// ---- DUTs/IO/PDOs/InfoData_6F19DB2B.TcDUT
{attribute 'GeneratedUsingTerminal: EK1100-0000-0018'}
{attribute addProperty BoxType "EK1100-0000-0018"}
{attribute addProperty Id "StateAT %I*UINT2"}
{attribute addProperty CRC "1863965483"}
{attribute addProperty Size "2"}
TYPE InfoData_6F19DB2B :
STRUCT
	{attribute addProperty Name "State"}
	State AT %I* : UINT;
END_STRUCT
END_TYPE

// ---- DUTs/IO/PDOs/YVR_Inputs_4719D0DB.TcDUT
{attribute 'GeneratedUsingTerminal: APS1003-7000-0016'}
{attribute addProperty BoxType "APS1003-7000-0016"}
{attribute addProperty Id "StatusWordAT %I*UINT2Current_D_0X0AT %I*INT2Current_D_0X1AT %I*INT2Current_D_0X2AT %I*INT2Current_D_0Y0AT %I*INT2Current_D_0Y1AT %I*INT2Current_D_0Y2AT %I*INT2Current_D_1X0AT %I*INT2Current_D_1X1AT %I*INT2Current_D_1X2AT %I*INT2Current_D_1Y0AT %I*INT2Current_D_1Y1AT %I*INT2Current_D_1Y2AT %I*INT2Current_D_2X0AT %I*INT2Current_D_2X1AT %I*INT2Current_D_2X2AT %I*INT2Current_D_2Y0AT %I*INT2Current_D_2Y1AT %I*INT2Current_D_2Y2AT %I*INT2Current_D_3X0AT %I*INT2Current_D_3X1AT %I*INT2Current_D_3X2AT %I*INT2Current_D_3Y0AT %I*INT2Current_D_3Y1AT %I*INT2Current_D_3Y2AT %I*INT2Current_Q_0X0AT %I*INT2Current_Q_0X1AT %I*INT2Current_Q_0X2AT %I*INT2Current_Q_0Y0AT %I*INT2Current_Q_0Y1AT %I*INT2Current_Q_0Y2AT %I*INT2Current_Q_1X0AT %I*INT2Current_Q_1X1AT %I*INT2Current_Q_1X2AT %I*INT2Current_Q_1Y0AT %I*INT2Current_Q_1Y1AT %I*INT2Current_Q_1Y2AT %I*INT2Current_Q_2X0AT %I*INT2Current_Q_2X1AT %I*INT2Current_Q_2X2AT %I*INT2Current_Q_2Y0AT %I*INT2Current_Q_2Y1AT %I*INT2Current_Q_2Y2AT %I*INT2Current_Q_3X0AT %I*INT2Current_Q_3X1AT %I*INT2Current_Q_3X2AT %I*INT2Current_Q_3Y0AT %I*INT2Current_Q_3Y1AT %I*INT2Current_Q_3Y2AT %I*INT2"}
{attribute addProperty CRC "1192874203"}
{attribute addProperty Size "98"}
TYPE YVR_Inputs_4719D0DB EXTENDS InputBase_8311D824 :
STRUCT
	{attribute addProperty Name "StatusWord"}
	StatusWord AT %I* : UINT;
	{attribute addProperty Name "Current_D_0X0"}
	Current_D_0X0 AT %I* : INT;
	{attribute addProperty Name "Current_D_0X1"}
	Current_D_0X1 AT %I* : INT;
	{attribute addProperty Name "Current_D_0X2"}
	Current_D_0X2 AT %I* : INT;
	{attribute addProperty Name "Current_D_0Y0"}
	Current_D_0Y0 AT %I* : INT;
	{attribute addProperty Name "Current_D_0Y1"}
	Current_D_0Y1 AT %I* : INT;
	{attribute addProperty Name "Current_D_0Y2"}
	Current_D_0Y2 AT %I* : INT;
	{attribute addProperty Name "Current_D_1X0"}
	Current_D_1X0 AT %I* : INT;
	{attribute addProperty Name "Current_D_1X1"}
	Current_D_1X1 AT %I* : INT;
	{attribute addProperty Name "Current_D_1X2"}
	Current_D_1X2 AT %I* : INT;
	{attribute addProperty Name "Current_D_1Y0"}
	Current_D_1Y0 AT %I* : INT;
	{attribute addProperty Name "Current_D_1Y1"}
	Current_D_1Y1 AT %I* : INT;
	{attribute addProperty Name "Current_D_1Y2"}
	Current_D_1Y2 AT %I* : INT;
	{attribute addProperty Name "Current_D_2X0"}
	Current_D_2X0 AT %I* : INT;
	{attribute addProperty Name "Current_D_2X1"}
	Current_D_2X1 AT %I* : INT;
	{attribute addProperty Name "Current_D_2X2"}
	Current_D_2X2 AT %I* : INT;
	{attribute addProperty Name "Current_D_2Y0"}
	Current_D_2Y0 AT %I* : INT;
	{attribute addProperty Name "Current_D_2Y1"}
	Current_D_2Y1 AT %I* : INT;
	{attribute addProperty Name "Current_D_2Y2"}
	Current_D_2Y2 AT %I* : INT;
	{attribute addProperty Name "Current_D_3X0"}
	Current_D_3X0 AT %I* : INT;
	{attribute addProperty Name "Current_D_3X1"}
	Current_D_3X1 AT %I* : INT;
	{attribute addProperty Name "Current_D_3X2"}
	Current_D_3X2 AT %I* : INT;
	{attribute addProperty Name "Current_D_3Y0"}
	Current_D_3Y0 AT %I* : INT;
	{attribute addProperty Name "Current_D_3Y1"}
	Current_D_3Y1 AT %I* : INT;
	{attribute addProperty Name "Current_D_3Y2"}
	Current_D_3Y2 AT %I* : INT;
	{attribute addProperty Name "Current_Q_0X0"}
	Current_Q_0X0 AT %I* : INT;
	{attribute addProperty Name "Current_Q_0X1"}
	Current_Q_0X1 AT %I* : INT;
	{attribute addProperty Name "Current_Q_0X2"}
	Current_Q_0X2 AT %I* : INT;
	{attribute addProperty Name "Current_Q_0Y0"}
	Current_Q_0Y0 AT %I* : INT;
	{attribute addProperty Name "Current_Q_0Y1"}
	Current_Q_0Y1 AT %I* : INT;
	{attribute addProperty Name "Current_Q_0Y2"}
	Current_Q_0Y2 AT %I* : INT;
	{attribute addProperty Name "Current_Q_1X0"}
	Current_Q_1X0 AT %I* : INT;
	{attribute addProperty Name "Current_Q_1X1"}
	Current_Q_1X1 AT %I* : INT;
	{attribute addProperty Name "Current_Q_1X2"}
	Current_Q_1X2 AT %I* : INT;
	{attribute addProperty Name "Current_Q_1Y0"}
	Current_Q_1Y0 AT %I* : INT;
	{attribute addProperty Name "Current_Q_1Y1"}
	Current_Q_1Y1 AT %I* : INT;
	{attribute addProperty Name "Current_Q_1Y2"}
	Current_Q_1Y2 AT %I* : INT;
	{attribute addProperty Name "Current_Q_2X0"}
	Current_Q_2X0 AT %I* : INT;
	{attribute addProperty Name "Current_Q_2X1"}
	Current_Q_2X1 AT %I* : INT;
	{attribute addProperty Name "Current_Q_2X2"}
	Current_Q_2X2 AT %I* : INT;
	{attribute addProperty Name "Current_Q_2Y0"}
	Current_Q_2Y0 AT %I* : INT;
	{attribute addProperty Name "Current_Q_2Y1"}
	Current_Q_2Y1 AT %I* : INT;
	{attribute addProperty Name "Current_Q_2Y2"}
	Current_Q_2Y2 AT %I* : INT;
	{attribute addProperty Name "Current_Q_3X0"}
	Current_Q_3X0 AT %I* : INT;
	{attribute addProperty Name "Current_Q_3X1"}
	Current_Q_3X1 AT %I* : INT;
	{attribute addProperty Name "Current_Q_3X2"}
	Current_Q_3X2 AT %I* : INT;
	{attribute addProperty Name "Current_Q_3Y0"}
	Current_Q_3Y0 AT %I* : INT;
	{attribute addProperty Name "Current_Q_3Y1"}
	Current_Q_3Y1 AT %I* : INT;
	{attribute addProperty Name "Current_Q_3Y2"}
	Current_Q_3Y2 AT %I* : INT;
END_STRUCT
END_TYPE

// ---- DUTs/IO/PDOs/YVR_Outputs_31F2CBB3.TcDUT
{attribute 'GeneratedUsingTerminal: APS1003-7000-0016'}
{attribute addProperty BoxType "APS1003-7000-0016"}
{attribute addProperty Id "ControlWordAT %Q*UINT2Current_D_0X0AT %Q*INT2Current_D_0X1AT %Q*INT2Current_D_0X2AT %Q*INT2Current_D_0Y0AT %Q*INT2Current_D_0Y1AT %Q*INT2Current_D_0Y2AT %Q*INT2Current_D_1X0AT %Q*INT2Current_D_1X1AT %Q*INT2Current_D_1X2AT %Q*INT2Current_D_1Y0AT %Q*INT2Current_D_1Y1AT %Q*INT2Current_D_1Y2AT %Q*INT2Current_D_2X0AT %Q*INT2Current_D_2X1AT %Q*INT2Current_D_2X2AT %Q*INT2Current_D_2Y0AT %Q*INT2Current_D_2Y1AT %Q*INT2Current_D_2Y2AT %Q*INT2Current_D_3X0AT %Q*INT2Current_D_3X1AT %Q*INT2Current_D_3X2AT %Q*INT2Current_D_3Y0AT %Q*INT2Current_D_3Y1AT %Q*INT2Current_D_3Y2AT %Q*INT2Current_Q_0X0AT %Q*INT2Current_Q_0X1AT %Q*INT2Current_Q_0X2AT %Q*INT2Current_Q_0Y0AT %Q*INT2Current_Q_0Y1AT %Q*INT2Current_Q_0Y2AT %Q*INT2Current_Q_1X0AT %Q*INT2Current_Q_1X1AT %Q*INT2Current_Q_1X2AT %Q*INT2Current_Q_1Y0AT %Q*INT2Current_Q_1Y1AT %Q*INT2Current_Q_1Y2AT %Q*INT2Current_Q_2X0AT %Q*INT2Current_Q_2X1AT %Q*INT2Current_Q_2X2AT %Q*INT2Current_Q_2Y0AT %Q*INT2Current_Q_2Y1AT %Q*INT2Current_Q_2Y2AT %Q*INT2Current_Q_3X0AT %Q*INT2Current_Q_3X1AT %Q*INT2Current_Q_3X2AT %Q*INT2Current_Q_3Y0AT %Q*INT2Current_Q_3Y1AT %Q*INT2Current_Q_3Y2AT %Q*INT2PhiE_0X0AT %Q*UINT2PhiE_0X1AT %Q*UINT2PhiE_0X2AT %Q*UINT2PhiE_0Y0AT %Q*UINT2PhiE_0Y1AT %Q*UINT2PhiE_0Y2AT %Q*UINT2PhiE_1X0AT %Q*UINT2PhiE_1X1AT %Q*UINT2PhiE_1X2AT %Q*UINT2PhiE_1Y0AT %Q*UINT2PhiE_1Y1AT %Q*UINT2PhiE_1Y2AT %Q*UINT2PhiE_2X0AT %Q*UINT2PhiE_2X1AT %Q*UINT2PhiE_2X2AT %Q*UINT2PhiE_2Y0AT %Q*UINT2PhiE_2Y1AT %Q*UINT2PhiE_2Y2AT %Q*UINT2PhiE_3X0AT %Q*UINT2PhiE_3X1AT %Q*UINT2PhiE_3X2AT %Q*UINT2PhiE_3Y0AT %Q*UINT2PhiE_3Y1AT %Q*UINT2PhiE_3Y2AT %Q*UINT2"}
{attribute addProperty CRC "837995443"}
{attribute addProperty Size "146"}
TYPE YVR_Outputs_31F2CBB3 EXTENDS OutputBase_10CEE7DE :
STRUCT
	{attribute addProperty Name "ControlWord"}
	ControlWord AT %Q* : UINT;
	{attribute addProperty Name "Current_D_0X0"}
	Current_D_0X0 AT %Q* : INT;
	{attribute addProperty Name "Current_D_0X1"}
	Current_D_0X1 AT %Q* : INT;
	{attribute addProperty Name "Current_D_0X2"}
	Current_D_0X2 AT %Q* : INT;
	{attribute addProperty Name "Current_D_0Y0"}
	Current_D_0Y0 AT %Q* : INT;
	{attribute addProperty Name "Current_D_0Y1"}
	Current_D_0Y1 AT %Q* : INT;
	{attribute addProperty Name "Current_D_0Y2"}
	Current_D_0Y2 AT %Q* : INT;
	{attribute addProperty Name "Current_D_1X0"}
	Current_D_1X0 AT %Q* : INT;
	{attribute addProperty Name "Current_D_1X1"}
	Current_D_1X1 AT %Q* : INT;
	{attribute addProperty Name "Current_D_1X2"}
	Current_D_1X2 AT %Q* : INT;
	{attribute addProperty Name "Current_D_1Y0"}
	Current_D_1Y0 AT %Q* : INT;
	{attribute addProperty Name "Current_D_1Y1"}
	Current_D_1Y1 AT %Q* : INT;
	{attribute addProperty Name "Current_D_1Y2"}
	Current_D_1Y2 AT %Q* : INT;
	{attribute addProperty Name "Current_D_2X0"}
	Current_D_2X0 AT %Q* : INT;
	{attribute addProperty Name "Current_D_2X1"}
	Current_D_2X1 AT %Q* : INT;
	{attribute addProperty Name "Current_D_2X2"}
	Current_D_2X2 AT %Q* : INT;
	{attribute addProperty Name "Current_D_2Y0"}
	Current_D_2Y0 AT %Q* : INT;
	{attribute addProperty Name "Current_D_2Y1"}
	Current_D_2Y1 AT %Q* : INT;
	{attribute addProperty Name "Current_D_2Y2"}
	Current_D_2Y2 AT %Q* : INT;
	{attribute addProperty Name "Current_D_3X0"}
	Current_D_3X0 AT %Q* : INT;
	{attribute addProperty Name "Current_D_3X1"}
	Current_D_3X1 AT %Q* : INT;
	{attribute addProperty Name "Current_D_3X2"}
	Current_D_3X2 AT %Q* : INT;
	{attribute addProperty Name "Current_D_3Y0"}
	Current_D_3Y0 AT %Q* : INT;
	{attribute addProperty Name "Current_D_3Y1"}
	Current_D_3Y1 AT %Q* : INT;
	{attribute addProperty Name "Current_D_3Y2"}
	Current_D_3Y2 AT %Q* : INT;
	{attribute addProperty Name "Current_Q_0X0"}
	Current_Q_0X0 AT %Q* : INT;
	{attribute addProperty Name "Current_Q_0X1"}
	Current_Q_0X1 AT %Q* : INT;
	{attribute addProperty Name "Current_Q_0X2"}
	Current_Q_0X2 AT %Q* : INT;
	{attribute addProperty Name "Current_Q_0Y0"}
	Current_Q_0Y0 AT %Q* : INT;
	{attribute addProperty Name "Current_Q_0Y1"}
	Current_Q_0Y1 AT %Q* : INT;
	{attribute addProperty Name "Current_Q_0Y2"}
	Current_Q_0Y2 AT %Q* : INT;
	{attribute addProperty Name "Current_Q_1X0"}
	Current_Q_1X0 AT %Q* : INT;
	{attribute addProperty Name "Current_Q_1X1"}
	Current_Q_1X1 AT %Q* : INT;
	{attribute addProperty Name "Current_Q_1X2"}
	Current_Q_1X2 AT %Q* : INT;
	{attribute addProperty Name "Current_Q_1Y0"}
	Current_Q_1Y0 AT %Q* : INT;
	{attribute addProperty Name "Current_Q_1Y1"}
	Current_Q_1Y1 AT %Q* : INT;
	{attribute addProperty Name "Current_Q_1Y2"}
	Current_Q_1Y2 AT %Q* : INT;
	{attribute addProperty Name "Current_Q_2X0"}
	Current_Q_2X0 AT %Q* : INT;
	{attribute addProperty Name "Current_Q_2X1"}
	Current_Q_2X1 AT %Q* : INT;
	{attribute addProperty Name "Current_Q_2X2"}
	Current_Q_2X2 AT %Q* : INT;
	{attribute addProperty Name "Current_Q_2Y0"}
	Current_Q_2Y0 AT %Q* : INT;
	{attribute addProperty Name "Current_Q_2Y1"}
	Current_Q_2Y1 AT %Q* : INT;
	{attribute addProperty Name "Current_Q_2Y2"}
	Current_Q_2Y2 AT %Q* : INT;
	{attribute addProperty Name "Current_Q_3X0"}
	Current_Q_3X0 AT %Q* : INT;
	{attribute addProperty Name "Current_Q_3X1"}
	Current_Q_3X1 AT %Q* : INT;
	{attribute addProperty Name "Current_Q_3X2"}
	Current_Q_3X2 AT %Q* : INT;
	{attribute addProperty Name "Current_Q_3Y0"}
	Current_Q_3Y0 AT %Q* : INT;
	{attribute addProperty Name "Current_Q_3Y1"}
	Current_Q_3Y1 AT %Q* : INT;
	{attribute addProperty Name "Current_Q_3Y2"}
	Current_Q_3Y2 AT %Q* : INT;
	{attribute addProperty Name "PhiE_0X0"}
	PhiE_0X0 AT %Q* : UINT;
	{attribute addProperty Name "PhiE_0X1"}
	PhiE_0X1 AT %Q* : UINT;
	{attribute addProperty Name "PhiE_0X2"}
	PhiE_0X2 AT %Q* : UINT;
	{attribute addProperty Name "PhiE_0Y0"}
	PhiE_0Y0 AT %Q* : UINT;
	{attribute addProperty Name "PhiE_0Y1"}
	PhiE_0Y1 AT %Q* : UINT;
	{attribute addProperty Name "PhiE_0Y2"}
	PhiE_0Y2 AT %Q* : UINT;
	{attribute addProperty Name "PhiE_1X0"}
	PhiE_1X0 AT %Q* : UINT;
	{attribute addProperty Name "PhiE_1X1"}
	PhiE_1X1 AT %Q* : UINT;
	{attribute addProperty Name "PhiE_1X2"}
	PhiE_1X2 AT %Q* : UINT;
	{attribute addProperty Name "PhiE_1Y0"}
	PhiE_1Y0 AT %Q* : UINT;
	{attribute addProperty Name "PhiE_1Y1"}
	PhiE_1Y1 AT %Q* : UINT;
	{attribute addProperty Name "PhiE_1Y2"}
	PhiE_1Y2 AT %Q* : UINT;
	{attribute addProperty Name "PhiE_2X0"}
	PhiE_2X0 AT %Q* : UINT;
	{attribute addProperty Name "PhiE_2X1"}
	PhiE_2X1 AT %Q* : UINT;
	{attribute addProperty Name "PhiE_2X2"}
	PhiE_2X2 AT %Q* : UINT;
	{attribute addProperty Name "PhiE_2Y0"}
	PhiE_2Y0 AT %Q* : UINT;
	{attribute addProperty Name "PhiE_2Y1"}
	PhiE_2Y1 AT %Q* : UINT;
	{attribute addProperty Name "PhiE_2Y2"}
	PhiE_2Y2 AT %Q* : UINT;
	{attribute addProperty Name "PhiE_3X0"}
	PhiE_3X0 AT %Q* : UINT;
	{attribute addProperty Name "PhiE_3X1"}
	PhiE_3X1 AT %Q* : UINT;
	{attribute addProperty Name "PhiE_3X2"}
	PhiE_3X2 AT %Q* : UINT;
	{attribute addProperty Name "PhiE_3Y0"}
	PhiE_3Y0 AT %Q* : UINT;
	{attribute addProperty Name "PhiE_3Y1"}
	PhiE_3Y1 AT %Q* : UINT;
	{attribute addProperty Name "PhiE_3Y2"}
	PhiE_3Y2 AT %Q* : UINT;
END_STRUCT
END_TYPE

// ---- DUTs/IO/PDOs/WcState_9091E0EB.TcDUT
{attribute 'GeneratedUsingTerminal: APS1003-7000-0016'}
{attribute addProperty BoxType "APS1003-7000-0016"}
{attribute addProperty Id "WcStateAT %I*BOOL1InputToggleAT %I*BOOL1"}
{attribute addProperty CRC "2425479403"}
{attribute addProperty Size "2"}
TYPE WcState_9091E0EB :
STRUCT
	{attribute addProperty Name "WcState"}
	WcState AT %I* : BOOL;
	{attribute addProperty Name "InputToggle"}
	InputToggle AT %I* : BOOL;
END_STRUCT
END_TYPE

// ---- DUTs/IO/PDOs/InfoData_BEF6B88E.TcDUT
{attribute 'GeneratedUsingTerminal: APS1003-7000-0016'}
{attribute addProperty BoxType "APS1003-7000-0016"}
{attribute addProperty Id "AdsAddrAT %I*AMSADDR8DcOutputShiftAT %I*DINT4DcInputShiftAT %I*DINT4StateAT %I*UINT2"}
{attribute addProperty CRC "3203840142"}
{attribute addProperty Size "18"}
TYPE InfoData_BEF6B88E EXTENDS InputBase_8311D824 :
STRUCT
	{attribute addProperty Name "AdsAddr"}
	AdsAddr AT %I* : AMSADDR;
	{attribute addProperty Name "DcOutputShift"}
	DcOutputShift AT %I* : DINT;
	{attribute addProperty Name "DcInputShift"}
	DcInputShift AT %I* : DINT;
	{attribute addProperty Name "State"}
	State AT %I* : UINT;
END_STRUCT
END_TYPE

// ---- DUTs/IO/PDOs/FB_Inputs_F0F03BDD.TcDUT
{attribute 'GeneratedUsingTerminal: APS1003-5000-0016'}
{attribute addProperty BoxType "APS1003-5000-0016"}
{attribute addProperty Id "StatusAT %I*LWORD8A0_X_FieldAT %I*INT2A0_Y_FieldAT %I*INT2A0_Z_FieldAT %I*INT2A2_X_FieldAT %I*INT2A2_Y_FieldAT %I*INT2A2_Z_FieldAT %I*INT2A4_X_FieldAT %I*INT2A4_Y_FieldAT %I*INT2A4_Z_FieldAT %I*INT2A6_X_FieldAT %I*INT2A6_Y_FieldAT %I*INT2A6_Z_FieldAT %I*INT2A8_X_FieldAT %I*INT2A8_Y_FieldAT %I*INT2A8_Z_FieldAT %I*INT2B1_X_FieldAT %I*INT2B1_Y_FieldAT %I*INT2B1_Z_FieldAT %I*INT2B3_X_FieldAT %I*INT2B3_Y_FieldAT %I*INT2B3_Z_FieldAT %I*INT2B5_X_FieldAT %I*INT2B5_Y_FieldAT %I*INT2B5_Z_FieldAT %I*INT2B7_X_FieldAT %I*INT2B7_Y_FieldAT %I*INT2B7_Z_FieldAT %I*INT2B9_X_FieldAT %I*INT2B9_Y_FieldAT %I*INT2B9_Z_FieldAT %I*INT2C0_X_FieldAT %I*INT2C0_Y_FieldAT %I*INT2C0_Z_FieldAT %I*INT2C2_X_FieldAT %I*INT2C2_Y_FieldAT %I*INT2C2_Z_FieldAT %I*INT2C4_X_FieldAT %I*INT2C4_Y_FieldAT %I*INT2C4_Z_FieldAT %I*INT2C6_X_FieldAT %I*INT2C6_Y_FieldAT %I*INT2C6_Z_FieldAT %I*INT2C8_X_FieldAT %I*INT2C8_Y_FieldAT %I*INT2C8_Z_FieldAT %I*INT2D1_X_FieldAT %I*INT2D1_Y_FieldAT %I*INT2D1_Z_FieldAT %I*INT2D3_X_FieldAT %I*INT2D3_Y_FieldAT %I*INT2D3_Z_FieldAT %I*INT2D5_X_FieldAT %I*INT2D5_Y_FieldAT %I*INT2D5_Z_FieldAT %I*INT2D7_X_FieldAT %I*INT2D7_Y_FieldAT %I*INT2D7_Z_FieldAT %I*INT2D9_X_FieldAT %I*INT2D9_Y_FieldAT %I*INT2D9_Z_FieldAT %I*INT2E0_X_FieldAT %I*INT2E0_Y_FieldAT %I*INT2E0_Z_FieldAT %I*INT2E2_X_FieldAT %I*INT2E2_Y_FieldAT %I*INT2E2_Z_FieldAT %I*INT2E4_X_FieldAT %I*INT2E4_Y_FieldAT %I*INT2E4_Z_FieldAT %I*INT2E6_X_FieldAT %I*INT2E6_Y_FieldAT %I*INT2E6_Z_FieldAT %I*INT2E8_X_FieldAT %I*INT2E8_Y_FieldAT %I*INT2E8_Z_FieldAT %I*INT2F1_X_FieldAT %I*INT2F1_Y_FieldAT %I*INT2F1_Z_FieldAT %I*INT2F3_X_FieldAT %I*INT2F3_Y_FieldAT %I*INT2F3_Z_FieldAT %I*INT2F5_X_FieldAT %I*INT2F5_Y_FieldAT %I*INT2F5_Z_FieldAT %I*INT2F7_X_FieldAT %I*INT2F7_Y_FieldAT %I*INT2F7_Z_FieldAT %I*INT2F9_X_FieldAT %I*INT2F9_Y_FieldAT %I*INT2F9_Z_FieldAT %I*INT2G0_X_FieldAT %I*INT2G0_Y_FieldAT %I*INT2G0_Z_FieldAT %I*INT2G2_X_FieldAT %I*INT2G2_Y_FieldAT %I*INT2G2_Z_FieldAT %I*INT2G4_X_FieldAT %I*INT2G4_Y_FieldAT %I*INT2G4_Z_FieldAT %I*INT2G6_X_FieldAT %I*INT2G6_Y_FieldAT %I*INT2G6_Z_FieldAT %I*INT2G8_X_FieldAT %I*INT2G8_Y_FieldAT %I*INT2G8_Z_FieldAT %I*INT2H1_X_FieldAT %I*INT2H1_Y_FieldAT %I*INT2H1_Z_FieldAT %I*INT2H3_X_FieldAT %I*INT2H3_Y_FieldAT %I*INT2H3_Z_FieldAT %I*INT2H5_X_FieldAT %I*INT2H5_Y_FieldAT %I*INT2H5_Z_FieldAT %I*INT2H7_X_FieldAT %I*INT2H7_Y_FieldAT %I*INT2H7_Z_FieldAT %I*INT2H9_X_FieldAT %I*INT2H9_Y_FieldAT %I*INT2H9_Z_FieldAT %I*INT2I0_X_FieldAT %I*INT2I0_Y_FieldAT %I*INT2I0_Z_FieldAT %I*INT2I2_X_FieldAT %I*INT2I2_Y_FieldAT %I*INT2I2_Z_FieldAT %I*INT2I4_X_FieldAT %I*INT2I4_Y_FieldAT %I*INT2I4_Z_FieldAT %I*INT2I6_X_FieldAT %I*INT2I6_Y_FieldAT %I*INT2I6_Z_FieldAT %I*INT2I8_X_FieldAT %I*INT2I8_Y_FieldAT %I*INT2I8_Z_FieldAT %I*INT2J1_X_FieldAT %I*INT2J1_Y_FieldAT %I*INT2J1_Z_FieldAT %I*INT2J3_X_FieldAT %I*INT2J3_Y_FieldAT %I*INT2J3_Z_FieldAT %I*INT2J5_X_FieldAT %I*INT2J5_Y_FieldAT %I*INT2J5_Z_FieldAT %I*INT2J7_X_FieldAT %I*INT2J7_Y_FieldAT %I*INT2J7_Z_FieldAT %I*INT2J9_X_FieldAT %I*INT2J9_Y_FieldAT %I*INT2J9_Z_FieldAT %I*INT2"}
{attribute addProperty CRC "4042275805"}
{attribute addProperty Size "308"}
TYPE FB_Inputs_F0F03BDD EXTENDS InputBase_8311D824 :
STRUCT
	{attribute addProperty Name "Status"}
	Status AT %I* : LWORD;
	{attribute addProperty Name "A0_X_Field"}
	A0_X_Field AT %I* : INT;
	{attribute addProperty Name "A0_Y_Field"}
	A0_Y_Field AT %I* : INT;
	{attribute addProperty Name "A0_Z_Field"}
	A0_Z_Field AT %I* : INT;
	{attribute addProperty Name "A2_X_Field"}
	A2_X_Field AT %I* : INT;
	{attribute addProperty Name "A2_Y_Field"}
	A2_Y_Field AT %I* : INT;
	{attribute addProperty Name "A2_Z_Field"}
	A2_Z_Field AT %I* : INT;
	{attribute addProperty Name "A4_X_Field"}
	A4_X_Field AT %I* : INT;
	{attribute addProperty Name "A4_Y_Field"}
	A4_Y_Field AT %I* : INT;
	{attribute addProperty Name "A4_Z_Field"}
	A4_Z_Field AT %I* : INT;
	{attribute addProperty Name "A6_X_Field"}
	A6_X_Field AT %I* : INT;
	{attribute addProperty Name "A6_Y_Field"}
	A6_Y_Field AT %I* : INT;
	{attribute addProperty Name "A6_Z_Field"}
	A6_Z_Field AT %I* : INT;
	{attribute addProperty Name "A8_X_Field"}
	A8_X_Field AT %I* : INT;
	{attribute addProperty Name "A8_Y_Field"}
	A8_Y_Field AT %I* : INT;
	{attribute addProperty Name "A8_Z_Field"}
	A8_Z_Field AT %I* : INT;
	{attribute addProperty Name "B1_X_Field"}
	B1_X_Field AT %I* : INT;
	{attribute addProperty Name "B1_Y_Field"}
	B1_Y_Field AT %I* : INT;
	{attribute addProperty Name "B1_Z_Field"}
	B1_Z_Field AT %I* : INT;
	{attribute addProperty Name "B3_X_Field"}
	B3_X_Field AT %I* : INT;
	{attribute addProperty Name "B3_Y_Field"}
	B3_Y_Field AT %I* : INT;
	{attribute addProperty Name "B3_Z_Field"}
	B3_Z_Field AT %I* : INT;
	{attribute addProperty Name "B5_X_Field"}
	B5_X_Field AT %I* : INT;
	{attribute addProperty Name "B5_Y_Field"}
	B5_Y_Field AT %I* : INT;
	{attribute addProperty Name "B5_Z_Field"}
	B5_Z_Field AT %I* : INT;
	{attribute addProperty Name "B7_X_Field"}
	B7_X_Field AT %I* : INT;
	{attribute addProperty Name "B7_Y_Field"}
	B7_Y_Field AT %I* : INT;
	{attribute addProperty Name "B7_Z_Field"}
	B7_Z_Field AT %I* : INT;
	{attribute addProperty Name "B9_X_Field"}
	B9_X_Field AT %I* : INT;
	{attribute addProperty Name "B9_Y_Field"}
	B9_Y_Field AT %I* : INT;
	{attribute addProperty Name "B9_Z_Field"}
	B9_Z_Field AT %I* : INT;
	{attribute addProperty Name "C0_X_Field"}
	C0_X_Field AT %I* : INT;
	{attribute addProperty Name "C0_Y_Field"}
	C0_Y_Field AT %I* : INT;
	{attribute addProperty Name "C0_Z_Field"}
	C0_Z_Field AT %I* : INT;
	{attribute addProperty Name "C2_X_Field"}
	C2_X_Field AT %I* : INT;
	{attribute addProperty Name "C2_Y_Field"}
	C2_Y_Field AT %I* : INT;
	{attribute addProperty Name "C2_Z_Field"}
	C2_Z_Field AT %I* : INT;
	{attribute addProperty Name "C4_X_Field"}
	C4_X_Field AT %I* : INT;
	{attribute addProperty Name "C4_Y_Field"}
	C4_Y_Field AT %I* : INT;
	{attribute addProperty Name "C4_Z_Field"}
	C4_Z_Field AT %I* : INT;
	{attribute addProperty Name "C6_X_Field"}
	C6_X_Field AT %I* : INT;
	{attribute addProperty Name "C6_Y_Field"}
	C6_Y_Field AT %I* : INT;
	{attribute addProperty Name "C6_Z_Field"}
	C6_Z_Field AT %I* : INT;
	{attribute addProperty Name "C8_X_Field"}
	C8_X_Field AT %I* : INT;
	{attribute addProperty Name "C8_Y_Field"}
	C8_Y_Field AT %I* : INT;
	{attribute addProperty Name "C8_Z_Field"}
	C8_Z_Field AT %I* : INT;
	{attribute addProperty Name "D1_X_Field"}
	D1_X_Field AT %I* : INT;
	{attribute addProperty Name "D1_Y_Field"}
	D1_Y_Field AT %I* : INT;
	{attribute addProperty Name "D1_Z_Field"}
	D1_Z_Field AT %I* : INT;
	{attribute addProperty Name "D3_X_Field"}
	D3_X_Field AT %I* : INT;
	{attribute addProperty Name "D3_Y_Field"}
	D3_Y_Field AT %I* : INT;
	{attribute addProperty Name "D3_Z_Field"}
	D3_Z_Field AT %I* : INT;
	{attribute addProperty Name "D5_X_Field"}
	D5_X_Field AT %I* : INT;
	{attribute addProperty Name "D5_Y_Field"}
	D5_Y_Field AT %I* : INT;
	{attribute addProperty Name "D5_Z_Field"}
	D5_Z_Field AT %I* : INT;
	{attribute addProperty Name "D7_X_Field"}
	D7_X_Field AT %I* : INT;
	{attribute addProperty Name "D7_Y_Field"}
	D7_Y_Field AT %I* : INT;
	{attribute addProperty Name "D7_Z_Field"}
	D7_Z_Field AT %I* : INT;
	{attribute addProperty Name "D9_X_Field"}
	D9_X_Field AT %I* : INT;
	{attribute addProperty Name "D9_Y_Field"}
	D9_Y_Field AT %I* : INT;
	{attribute addProperty Name "D9_Z_Field"}
	D9_Z_Field AT %I* : INT;
	{attribute addProperty Name "E0_X_Field"}
	E0_X_Field AT %I* : INT;
	{attribute addProperty Name "E0_Y_Field"}
	E0_Y_Field AT %I* : INT;
	{attribute addProperty Name "E0_Z_Field"}
	E0_Z_Field AT %I* : INT;
	{attribute addProperty Name "E2_X_Field"}
	E2_X_Field AT %I* : INT;
	{attribute addProperty Name "E2_Y_Field"}
	E2_Y_Field AT %I* : INT;
	{attribute addProperty Name "E2_Z_Field"}
	E2_Z_Field AT %I* : INT;
	{attribute addProperty Name "E4_X_Field"}
	E4_X_Field AT %I* : INT;
	{attribute addProperty Name "E4_Y_Field"}
	E4_Y_Field AT %I* : INT;
	{attribute addProperty Name "E4_Z_Field"}
	E4_Z_Field AT %I* : INT;
	{attribute addProperty Name "E6_X_Field"}
	E6_X_Field AT %I* : INT;
	{attribute addProperty Name "E6_Y_Field"}
	E6_Y_Field AT %I* : INT;
	{attribute addProperty Name "E6_Z_Field"}
	E6_Z_Field AT %I* : INT;
	{attribute addProperty Name "E8_X_Field"}
	E8_X_Field AT %I* : INT;
	{attribute addProperty Name "E8_Y_Field"}
	E8_Y_Field AT %I* : INT;
	{attribute addProperty Name "E8_Z_Field"}
	E8_Z_Field AT %I* : INT;
	{attribute addProperty Name "F1_X_Field"}
	F1_X_Field AT %I* : INT;
	{attribute addProperty Name "F1_Y_Field"}
	F1_Y_Field AT %I* : INT;
	{attribute addProperty Name "F1_Z_Field"}
	F1_Z_Field AT %I* : INT;
	{attribute addProperty Name "F3_X_Field"}
	F3_X_Field AT %I* : INT;
	{attribute addProperty Name "F3_Y_Field"}
	F3_Y_Field AT %I* : INT;
	{attribute addProperty Name "F3_Z_Field"}
	F3_Z_Field AT %I* : INT;
	{attribute addProperty Name "F5_X_Field"}
	F5_X_Field AT %I* : INT;
	{attribute addProperty Name "F5_Y_Field"}
	F5_Y_Field AT %I* : INT;
	{attribute addProperty Name "F5_Z_Field"}
	F5_Z_Field AT %I* : INT;
	{attribute addProperty Name "F7_X_Field"}
	F7_X_Field AT %I* : INT;
	{attribute addProperty Name "F7_Y_Field"}
	F7_Y_Field AT %I* : INT;
	{attribute addProperty Name "F7_Z_Field"}
	F7_Z_Field AT %I* : INT;
	{attribute addProperty Name "F9_X_Field"}
	F9_X_Field AT %I* : INT;
	{attribute addProperty Name "F9_Y_Field"}
	F9_Y_Field AT %I* : INT;
	{attribute addProperty Name "F9_Z_Field"}
	F9_Z_Field AT %I* : INT;
	{attribute addProperty Name "G0_X_Field"}
	G0_X_Field AT %I* : INT;
	{attribute addProperty Name "G0_Y_Field"}
	G0_Y_Field AT %I* : INT;
	{attribute addProperty Name "G0_Z_Field"}
	G0_Z_Field AT %I* : INT;
	{attribute addProperty Name "G2_X_Field"}
	G2_X_Field AT %I* : INT;
	{attribute addProperty Name "G2_Y_Field"}
	G2_Y_Field AT %I* : INT;
	{attribute addProperty Name "G2_Z_Field"}
	G2_Z_Field AT %I* : INT;
	{attribute addProperty Name "G4_X_Field"}
	G4_X_Field AT %I* : INT;
	{attribute addProperty Name "G4_Y_Field"}
	G4_Y_Field AT %I* : INT;
	{attribute addProperty Name "G4_Z_Field"}
	G4_Z_Field AT %I* : INT;
	{attribute addProperty Name "G6_X_Field"}
	G6_X_Field AT %I* : INT;
	{attribute addProperty Name "G6_Y_Field"}
	G6_Y_Field AT %I* : INT;
	{attribute addProperty Name "G6_Z_Field"}
	G6_Z_Field AT %I* : INT;
	{attribute addProperty Name "G8_X_Field"}
	G8_X_Field AT %I* : INT;
	{attribute addProperty Name "G8_Y_Field"}
	G8_Y_Field AT %I* : INT;
	{attribute addProperty Name "G8_Z_Field"}
	G8_Z_Field AT %I* : INT;
	{attribute addProperty Name "H1_X_Field"}
	H1_X_Field AT %I* : INT;
	{attribute addProperty Name "H1_Y_Field"}
	H1_Y_Field AT %I* : INT;
	{attribute addProperty Name "H1_Z_Field"}
	H1_Z_Field AT %I* : INT;
	{attribute addProperty Name "H3_X_Field"}
	H3_X_Field AT %I* : INT;
	{attribute addProperty Name "H3_Y_Field"}
	H3_Y_Field AT %I* : INT;
	{attribute addProperty Name "H3_Z_Field"}
	H3_Z_Field AT %I* : INT;
	{attribute addProperty Name "H5_X_Field"}
	H5_X_Field AT %I* : INT;
	{attribute addProperty Name "H5_Y_Field"}
	H5_Y_Field AT %I* : INT;
	{attribute addProperty Name "H5_Z_Field"}
	H5_Z_Field AT %I* : INT;
	{attribute addProperty Name "H7_X_Field"}
	H7_X_Field AT %I* : INT;
	{attribute addProperty Name "H7_Y_Field"}
	H7_Y_Field AT %I* : INT;
	{attribute addProperty Name "H7_Z_Field"}
	H7_Z_Field AT %I* : INT;
	{attribute addProperty Name "H9_X_Field"}
	H9_X_Field AT %I* : INT;
	{attribute addProperty Name "H9_Y_Field"}
	H9_Y_Field AT %I* : INT;
	{attribute addProperty Name "H9_Z_Field"}
	H9_Z_Field AT %I* : INT;
	{attribute addProperty Name "I0_X_Field"}
	I0_X_Field AT %I* : INT;
	{attribute addProperty Name "I0_Y_Field"}
	I0_Y_Field AT %I* : INT;
	{attribute addProperty Name "I0_Z_Field"}
	I0_Z_Field AT %I* : INT;
	{attribute addProperty Name "I2_X_Field"}
	I2_X_Field AT %I* : INT;
	{attribute addProperty Name "I2_Y_Field"}
	I2_Y_Field AT %I* : INT;
	{attribute addProperty Name "I2_Z_Field"}
	I2_Z_Field AT %I* : INT;
	{attribute addProperty Name "I4_X_Field"}
	I4_X_Field AT %I* : INT;
	{attribute addProperty Name "I4_Y_Field"}
	I4_Y_Field AT %I* : INT;
	{attribute addProperty Name "I4_Z_Field"}
	I4_Z_Field AT %I* : INT;
	{attribute addProperty Name "I6_X_Field"}
	I6_X_Field AT %I* : INT;
	{attribute addProperty Name "I6_Y_Field"}
	I6_Y_Field AT %I* : INT;
	{attribute addProperty Name "I6_Z_Field"}
	I6_Z_Field AT %I* : INT;
	{attribute addProperty Name "I8_X_Field"}
	I8_X_Field AT %I* : INT;
	{attribute addProperty Name "I8_Y_Field"}
	I8_Y_Field AT %I* : INT;
	{attribute addProperty Name "I8_Z_Field"}
	I8_Z_Field AT %I* : INT;
	{attribute addProperty Name "J1_X_Field"}
	J1_X_Field AT %I* : INT;
	{attribute addProperty Name "J1_Y_Field"}
	J1_Y_Field AT %I* : INT;
	{attribute addProperty Name "J1_Z_Field"}
	J1_Z_Field AT %I* : INT;
	{attribute addProperty Name "J3_X_Field"}
	J3_X_Field AT %I* : INT;
	{attribute addProperty Name "J3_Y_Field"}
	J3_Y_Field AT %I* : INT;
	{attribute addProperty Name "J3_Z_Field"}
	J3_Z_Field AT %I* : INT;
	{attribute addProperty Name "J5_X_Field"}
	J5_X_Field AT %I* : INT;
	{attribute addProperty Name "J5_Y_Field"}
	J5_Y_Field AT %I* : INT;
	{attribute addProperty Name "J5_Z_Field"}
	J5_Z_Field AT %I* : INT;
	{attribute addProperty Name "J7_X_Field"}
	J7_X_Field AT %I* : INT;
	{attribute addProperty Name "J7_Y_Field"}
	J7_Y_Field AT %I* : INT;
	{attribute addProperty Name "J7_Z_Field"}
	J7_Z_Field AT %I* : INT;
	{attribute addProperty Name "J9_X_Field"}
	J9_X_Field AT %I* : INT;
	{attribute addProperty Name "J9_Y_Field"}
	J9_Y_Field AT %I* : INT;
	{attribute addProperty Name "J9_Z_Field"}
	J9_Z_Field AT %I* : INT;
END_STRUCT
END_TYPE

// ---- DUTs/IO/PDOs/InfoData_A7436BC6.TcDUT
{attribute 'GeneratedUsingTerminal: APS1003-5000-0016'}
{attribute addProperty BoxType "APS1003-5000-0016"}
{attribute addProperty Id "DcOutputShiftAT %I*DINT4DcInputShiftAT %I*DINT4StateAT %I*UINT2"}
{attribute addProperty CRC "2806213574"}
{attribute addProperty Size "10"}
TYPE InfoData_A7436BC6 EXTENDS InputBase_8311D824 :
STRUCT
	{attribute addProperty Name "DcOutputShift"}
	DcOutputShift AT %I* : DINT;
	{attribute addProperty Name "DcInputShift"}
	DcInputShift AT %I* : DINT;
	{attribute addProperty Name "State"}
	State AT %I* : UINT;
END_STRUCT
END_TYPE

// ---- DUTs/IO/PDOs/APS_Inputs_4719D0DB.TcDUT
{attribute 'GeneratedUsingTerminal: APS4322-7000-0017'}
{attribute addProperty BoxType "APS4322-7000-0017"}
{attribute addProperty Id "StatusWordAT %I*UINT2Current_D_0X0AT %I*INT2Current_D_0X1AT %I*INT2Current_D_0X2AT %I*INT2Current_D_0Y0AT %I*INT2Current_D_0Y1AT %I*INT2Current_D_0Y2AT %I*INT2Current_D_1X0AT %I*INT2Current_D_1X1AT %I*INT2Current_D_1X2AT %I*INT2Current_D_1Y0AT %I*INT2Current_D_1Y1AT %I*INT2Current_D_1Y2AT %I*INT2Current_D_2X0AT %I*INT2Current_D_2X1AT %I*INT2Current_D_2X2AT %I*INT2Current_D_2Y0AT %I*INT2Current_D_2Y1AT %I*INT2Current_D_2Y2AT %I*INT2Current_D_3X0AT %I*INT2Current_D_3X1AT %I*INT2Current_D_3X2AT %I*INT2Current_D_3Y0AT %I*INT2Current_D_3Y1AT %I*INT2Current_D_3Y2AT %I*INT2Current_Q_0X0AT %I*INT2Current_Q_0X1AT %I*INT2Current_Q_0X2AT %I*INT2Current_Q_0Y0AT %I*INT2Current_Q_0Y1AT %I*INT2Current_Q_0Y2AT %I*INT2Current_Q_1X0AT %I*INT2Current_Q_1X1AT %I*INT2Current_Q_1X2AT %I*INT2Current_Q_1Y0AT %I*INT2Current_Q_1Y1AT %I*INT2Current_Q_1Y2AT %I*INT2Current_Q_2X0AT %I*INT2Current_Q_2X1AT %I*INT2Current_Q_2X2AT %I*INT2Current_Q_2Y0AT %I*INT2Current_Q_2Y1AT %I*INT2Current_Q_2Y2AT %I*INT2Current_Q_3X0AT %I*INT2Current_Q_3X1AT %I*INT2Current_Q_3X2AT %I*INT2Current_Q_3Y0AT %I*INT2Current_Q_3Y1AT %I*INT2Current_Q_3Y2AT %I*INT2"}
{attribute addProperty CRC "1192874203"}
{attribute addProperty Size "98"}
TYPE APS_Inputs_4719D0DB EXTENDS InputBase_8311D824 :
STRUCT
	{attribute addProperty Name "StatusWord"}
	StatusWord AT %I* : UINT;
	{attribute addProperty Name "Current_D_0X0"}
	Current_D_0X0 AT %I* : INT;
	{attribute addProperty Name "Current_D_0X1"}
	Current_D_0X1 AT %I* : INT;
	{attribute addProperty Name "Current_D_0X2"}
	Current_D_0X2 AT %I* : INT;
	{attribute addProperty Name "Current_D_0Y0"}
	Current_D_0Y0 AT %I* : INT;
	{attribute addProperty Name "Current_D_0Y1"}
	Current_D_0Y1 AT %I* : INT;
	{attribute addProperty Name "Current_D_0Y2"}
	Current_D_0Y2 AT %I* : INT;
	{attribute addProperty Name "Current_D_1X0"}
	Current_D_1X0 AT %I* : INT;
	{attribute addProperty Name "Current_D_1X1"}
	Current_D_1X1 AT %I* : INT;
	{attribute addProperty Name "Current_D_1X2"}
	Current_D_1X2 AT %I* : INT;
	{attribute addProperty Name "Current_D_1Y0"}
	Current_D_1Y0 AT %I* : INT;
	{attribute addProperty Name "Current_D_1Y1"}
	Current_D_1Y1 AT %I* : INT;
	{attribute addProperty Name "Current_D_1Y2"}
	Current_D_1Y2 AT %I* : INT;
	{attribute addProperty Name "Current_D_2X0"}
	Current_D_2X0 AT %I* : INT;
	{attribute addProperty Name "Current_D_2X1"}
	Current_D_2X1 AT %I* : INT;
	{attribute addProperty Name "Current_D_2X2"}
	Current_D_2X2 AT %I* : INT;
	{attribute addProperty Name "Current_D_2Y0"}
	Current_D_2Y0 AT %I* : INT;
	{attribute addProperty Name "Current_D_2Y1"}
	Current_D_2Y1 AT %I* : INT;
	{attribute addProperty Name "Current_D_2Y2"}
	Current_D_2Y2 AT %I* : INT;
	{attribute addProperty Name "Current_D_3X0"}
	Current_D_3X0 AT %I* : INT;
	{attribute addProperty Name "Current_D_3X1"}
	Current_D_3X1 AT %I* : INT;
	{attribute addProperty Name "Current_D_3X2"}
	Current_D_3X2 AT %I* : INT;
	{attribute addProperty Name "Current_D_3Y0"}
	Current_D_3Y0 AT %I* : INT;
	{attribute addProperty Name "Current_D_3Y1"}
	Current_D_3Y1 AT %I* : INT;
	{attribute addProperty Name "Current_D_3Y2"}
	Current_D_3Y2 AT %I* : INT;
	{attribute addProperty Name "Current_Q_0X0"}
	Current_Q_0X0 AT %I* : INT;
	{attribute addProperty Name "Current_Q_0X1"}
	Current_Q_0X1 AT %I* : INT;
	{attribute addProperty Name "Current_Q_0X2"}
	Current_Q_0X2 AT %I* : INT;
	{attribute addProperty Name "Current_Q_0Y0"}
	Current_Q_0Y0 AT %I* : INT;
	{attribute addProperty Name "Current_Q_0Y1"}
	Current_Q_0Y1 AT %I* : INT;
	{attribute addProperty Name "Current_Q_0Y2"}
	Current_Q_0Y2 AT %I* : INT;
	{attribute addProperty Name "Current_Q_1X0"}
	Current_Q_1X0 AT %I* : INT;
	{attribute addProperty Name "Current_Q_1X1"}
	Current_Q_1X1 AT %I* : INT;
	{attribute addProperty Name "Current_Q_1X2"}
	Current_Q_1X2 AT %I* : INT;
	{attribute addProperty Name "Current_Q_1Y0"}
	Current_Q_1Y0 AT %I* : INT;
	{attribute addProperty Name "Current_Q_1Y1"}
	Current_Q_1Y1 AT %I* : INT;
	{attribute addProperty Name "Current_Q_1Y2"}
	Current_Q_1Y2 AT %I* : INT;
	{attribute addProperty Name "Current_Q_2X0"}
	Current_Q_2X0 AT %I* : INT;
	{attribute addProperty Name "Current_Q_2X1"}
	Current_Q_2X1 AT %I* : INT;
	{attribute addProperty Name "Current_Q_2X2"}
	Current_Q_2X2 AT %I* : INT;
	{attribute addProperty Name "Current_Q_2Y0"}
	Current_Q_2Y0 AT %I* : INT;
	{attribute addProperty Name "Current_Q_2Y1"}
	Current_Q_2Y1 AT %I* : INT;
	{attribute addProperty Name "Current_Q_2Y2"}
	Current_Q_2Y2 AT %I* : INT;
	{attribute addProperty Name "Current_Q_3X0"}
	Current_Q_3X0 AT %I* : INT;
	{attribute addProperty Name "Current_Q_3X1"}
	Current_Q_3X1 AT %I* : INT;
	{attribute addProperty Name "Current_Q_3X2"}
	Current_Q_3X2 AT %I* : INT;
	{attribute addProperty Name "Current_Q_3Y0"}
	Current_Q_3Y0 AT %I* : INT;
	{attribute addProperty Name "Current_Q_3Y1"}
	Current_Q_3Y1 AT %I* : INT;
	{attribute addProperty Name "Current_Q_3Y2"}
	Current_Q_3Y2 AT %I* : INT;
END_STRUCT
END_TYPE

// ---- DUTs/IO/PDOs/APS_Diagdata_CE5B986F.TcDUT
{attribute 'GeneratedUsingTerminal: APS4322-7000-0017'}
{attribute addProperty BoxType "APS4322-7000-0017"}
{attribute addProperty Id "DC_Link_VoltageAT %I*UINT2Power_supply_currentAT %I*INT2"}
{attribute addProperty CRC "3462109295"}
{attribute addProperty Size "4"}
TYPE APS_Diagdata_CE5B986F EXTENDS InputBase_8311D824 :
STRUCT
	{attribute addProperty Name "DC_Link_Voltage"}
	DC_Link_Voltage AT %I* : UINT;
	{attribute addProperty Name "Power_supply_current"}
	Power_supply_current AT %I* : INT;
END_STRUCT
END_TYPE

// ---- DUTs/IO/PDOs/APS_Comm_Inputs_388FE28E.TcDUT
{attribute 'GeneratedUsingTerminal: APS4322-7000-0017'}
{attribute addProperty BoxType "APS4322-7000-0017"}
{attribute addProperty Id "CommStatusWordAT %I*UINT2DataAT %I*ARRAY[0..3] OF UINT8"}
{attribute addProperty CRC "3146150883"}
{attribute addProperty Size "10"}
TYPE APS_Comm_Inputs_388FE28E EXTENDS InputBase_8311D824 :
STRUCT
	{attribute addProperty Name "CommStatusWord"}
	CommStatusWord AT %I* : UINT;
	{attribute addProperty Name "Data"}
	Data AT %I* : ARRAY[0..3] OF UINT;
END_STRUCT
END_TYPE

// ---- DUTs/IO/PDOs/APS_Outputs_31F2CBB3.TcDUT
{attribute 'GeneratedUsingTerminal: APS4322-7000-0017'}
{attribute addProperty BoxType "APS4322-7000-0017"}
{attribute addProperty Id "ControlWordAT %Q*UINT2Current_D_0X0AT %Q*INT2Current_D_0X1AT %Q*INT2Current_D_0X2AT %Q*INT2Current_D_0Y0AT %Q*INT2Current_D_0Y1AT %Q*INT2Current_D_0Y2AT %Q*INT2Current_D_1X0AT %Q*INT2Current_D_1X1AT %Q*INT2Current_D_1X2AT %Q*INT2Current_D_1Y0AT %Q*INT2Current_D_1Y1AT %Q*INT2Current_D_1Y2AT %Q*INT2Current_D_2X0AT %Q*INT2Current_D_2X1AT %Q*INT2Current_D_2X2AT %Q*INT2Current_D_2Y0AT %Q*INT2Current_D_2Y1AT %Q*INT2Current_D_2Y2AT %Q*INT2Current_D_3X0AT %Q*INT2Current_D_3X1AT %Q*INT2Current_D_3X2AT %Q*INT2Current_D_3Y0AT %Q*INT2Current_D_3Y1AT %Q*INT2Current_D_3Y2AT %Q*INT2Current_Q_0X0AT %Q*INT2Current_Q_0X1AT %Q*INT2Current_Q_0X2AT %Q*INT2Current_Q_0Y0AT %Q*INT2Current_Q_0Y1AT %Q*INT2Current_Q_0Y2AT %Q*INT2Current_Q_1X0AT %Q*INT2Current_Q_1X1AT %Q*INT2Current_Q_1X2AT %Q*INT2Current_Q_1Y0AT %Q*INT2Current_Q_1Y1AT %Q*INT2Current_Q_1Y2AT %Q*INT2Current_Q_2X0AT %Q*INT2Current_Q_2X1AT %Q*INT2Current_Q_2X2AT %Q*INT2Current_Q_2Y0AT %Q*INT2Current_Q_2Y1AT %Q*INT2Current_Q_2Y2AT %Q*INT2Current_Q_3X0AT %Q*INT2Current_Q_3X1AT %Q*INT2Current_Q_3X2AT %Q*INT2Current_Q_3Y0AT %Q*INT2Current_Q_3Y1AT %Q*INT2Current_Q_3Y2AT %Q*INT2PhiE_0X0AT %Q*UINT2PhiE_0X1AT %Q*UINT2PhiE_0X2AT %Q*UINT2PhiE_0Y0AT %Q*UINT2PhiE_0Y1AT %Q*UINT2PhiE_0Y2AT %Q*UINT2PhiE_1X0AT %Q*UINT2PhiE_1X1AT %Q*UINT2PhiE_1X2AT %Q*UINT2PhiE_1Y0AT %Q*UINT2PhiE_1Y1AT %Q*UINT2PhiE_1Y2AT %Q*UINT2PhiE_2X0AT %Q*UINT2PhiE_2X1AT %Q*UINT2PhiE_2X2AT %Q*UINT2PhiE_2Y0AT %Q*UINT2PhiE_2Y1AT %Q*UINT2PhiE_2Y2AT %Q*UINT2PhiE_3X0AT %Q*UINT2PhiE_3X1AT %Q*UINT2PhiE_3X2AT %Q*UINT2PhiE_3Y0AT %Q*UINT2PhiE_3Y1AT %Q*UINT2PhiE_3Y2AT %Q*UINT2"}
{attribute addProperty CRC "837995443"}
{attribute addProperty Size "146"}
TYPE APS_Outputs_31F2CBB3 EXTENDS OutputBase_10CEE7DE :
STRUCT
	{attribute addProperty Name "ControlWord"}
	ControlWord AT %Q* : UINT;
	{attribute addProperty Name "Current_D_0X0"}
	Current_D_0X0 AT %Q* : INT;
	{attribute addProperty Name "Current_D_0X1"}
	Current_D_0X1 AT %Q* : INT;
	{attribute addProperty Name "Current_D_0X2"}
	Current_D_0X2 AT %Q* : INT;
	{attribute addProperty Name "Current_D_0Y0"}
	Current_D_0Y0 AT %Q* : INT;
	{attribute addProperty Name "Current_D_0Y1"}
	Current_D_0Y1 AT %Q* : INT;
	{attribute addProperty Name "Current_D_0Y2"}
	Current_D_0Y2 AT %Q* : INT;
	{attribute addProperty Name "Current_D_1X0"}
	Current_D_1X0 AT %Q* : INT;
	{attribute addProperty Name "Current_D_1X1"}
	Current_D_1X1 AT %Q* : INT;
	{attribute addProperty Name "Current_D_1X2"}
	Current_D_1X2 AT %Q* : INT;
	{attribute addProperty Name "Current_D_1Y0"}
	Current_D_1Y0 AT %Q* : INT;
	{attribute addProperty Name "Current_D_1Y1"}
	Current_D_1Y1 AT %Q* : INT;
	{attribute addProperty Name "Current_D_1Y2"}
	Current_D_1Y2 AT %Q* : INT;
	{attribute addProperty Name "Current_D_2X0"}
	Current_D_2X0 AT %Q* : INT;
	{attribute addProperty Name "Current_D_2X1"}
	Current_D_2X1 AT %Q* : INT;
	{attribute addProperty Name "Current_D_2X2"}
	Current_D_2X2 AT %Q* : INT;
	{attribute addProperty Name "Current_D_2Y0"}
	Current_D_2Y0 AT %Q* : INT;
	{attribute addProperty Name "Current_D_2Y1"}
	Current_D_2Y1 AT %Q* : INT;
	{attribute addProperty Name "Current_D_2Y2"}
	Current_D_2Y2 AT %Q* : INT;
	{attribute addProperty Name "Current_D_3X0"}
	Current_D_3X0 AT %Q* : INT;
	{attribute addProperty Name "Current_D_3X1"}
	Current_D_3X1 AT %Q* : INT;
	{attribute addProperty Name "Current_D_3X2"}
	Current_D_3X2 AT %Q* : INT;
	{attribute addProperty Name "Current_D_3Y0"}
	Current_D_3Y0 AT %Q* : INT;
	{attribute addProperty Name "Current_D_3Y1"}
	Current_D_3Y1 AT %Q* : INT;
	{attribute addProperty Name "Current_D_3Y2"}
	Current_D_3Y2 AT %Q* : INT;
	{attribute addProperty Name "Current_Q_0X0"}
	Current_Q_0X0 AT %Q* : INT;
	{attribute addProperty Name "Current_Q_0X1"}
	Current_Q_0X1 AT %Q* : INT;
	{attribute addProperty Name "Current_Q_0X2"}
	Current_Q_0X2 AT %Q* : INT;
	{attribute addProperty Name "Current_Q_0Y0"}
	Current_Q_0Y0 AT %Q* : INT;
	{attribute addProperty Name "Current_Q_0Y1"}
	Current_Q_0Y1 AT %Q* : INT;
	{attribute addProperty Name "Current_Q_0Y2"}
	Current_Q_0Y2 AT %Q* : INT;
	{attribute addProperty Name "Current_Q_1X0"}
	Current_Q_1X0 AT %Q* : INT;
	{attribute addProperty Name "Current_Q_1X1"}
	Current_Q_1X1 AT %Q* : INT;
	{attribute addProperty Name "Current_Q_1X2"}
	Current_Q_1X2 AT %Q* : INT;
	{attribute addProperty Name "Current_Q_1Y0"}
	Current_Q_1Y0 AT %Q* : INT;
	{attribute addProperty Name "Current_Q_1Y1"}
	Current_Q_1Y1 AT %Q* : INT;
	{attribute addProperty Name "Current_Q_1Y2"}
	Current_Q_1Y2 AT %Q* : INT;
	{attribute addProperty Name "Current_Q_2X0"}
	Current_Q_2X0 AT %Q* : INT;
	{attribute addProperty Name "Current_Q_2X1"}
	Current_Q_2X1 AT %Q* : INT;
	{attribute addProperty Name "Current_Q_2X2"}
	Current_Q_2X2 AT %Q* : INT;
	{attribute addProperty Name "Current_Q_2Y0"}
	Current_Q_2Y0 AT %Q* : INT;
	{attribute addProperty Name "Current_Q_2Y1"}
	Current_Q_2Y1 AT %Q* : INT;
	{attribute addProperty Name "Current_Q_2Y2"}
	Current_Q_2Y2 AT %Q* : INT;
	{attribute addProperty Name "Current_Q_3X0"}
	Current_Q_3X0 AT %Q* : INT;
	{attribute addProperty Name "Current_Q_3X1"}
	Current_Q_3X1 AT %Q* : INT;
	{attribute addProperty Name "Current_Q_3X2"}
	Current_Q_3X2 AT %Q* : INT;
	{attribute addProperty Name "Current_Q_3Y0"}
	Current_Q_3Y0 AT %Q* : INT;
	{attribute addProperty Name "Current_Q_3Y1"}
	Current_Q_3Y1 AT %Q* : INT;
	{attribute addProperty Name "Current_Q_3Y2"}
	Current_Q_3Y2 AT %Q* : INT;
	{attribute addProperty Name "PhiE_0X0"}
	PhiE_0X0 AT %Q* : UINT;
	{attribute addProperty Name "PhiE_0X1"}
	PhiE_0X1 AT %Q* : UINT;
	{attribute addProperty Name "PhiE_0X2"}
	PhiE_0X2 AT %Q* : UINT;
	{attribute addProperty Name "PhiE_0Y0"}
	PhiE_0Y0 AT %Q* : UINT;
	{attribute addProperty Name "PhiE_0Y1"}
	PhiE_0Y1 AT %Q* : UINT;
	{attribute addProperty Name "PhiE_0Y2"}
	PhiE_0Y2 AT %Q* : UINT;
	{attribute addProperty Name "PhiE_1X0"}
	PhiE_1X0 AT %Q* : UINT;
	{attribute addProperty Name "PhiE_1X1"}
	PhiE_1X1 AT %Q* : UINT;
	{attribute addProperty Name "PhiE_1X2"}
	PhiE_1X2 AT %Q* : UINT;
	{attribute addProperty Name "PhiE_1Y0"}
	PhiE_1Y0 AT %Q* : UINT;
	{attribute addProperty Name "PhiE_1Y1"}
	PhiE_1Y1 AT %Q* : UINT;
	{attribute addProperty Name "PhiE_1Y2"}
	PhiE_1Y2 AT %Q* : UINT;
	{attribute addProperty Name "PhiE_2X0"}
	PhiE_2X0 AT %Q* : UINT;
	{attribute addProperty Name "PhiE_2X1"}
	PhiE_2X1 AT %Q* : UINT;
	{attribute addProperty Name "PhiE_2X2"}
	PhiE_2X2 AT %Q* : UINT;
	{attribute addProperty Name "PhiE_2Y0"}
	PhiE_2Y0 AT %Q* : UINT;
	{attribute addProperty Name "PhiE_2Y1"}
	PhiE_2Y1 AT %Q* : UINT;
	{attribute addProperty Name "PhiE_2Y2"}
	PhiE_2Y2 AT %Q* : UINT;
	{attribute addProperty Name "PhiE_3X0"}
	PhiE_3X0 AT %Q* : UINT;
	{attribute addProperty Name "PhiE_3X1"}
	PhiE_3X1 AT %Q* : UINT;
	{attribute addProperty Name "PhiE_3X2"}
	PhiE_3X2 AT %Q* : UINT;
	{attribute addProperty Name "PhiE_3Y0"}
	PhiE_3Y0 AT %Q* : UINT;
	{attribute addProperty Name "PhiE_3Y1"}
	PhiE_3Y1 AT %Q* : UINT;
	{attribute addProperty Name "PhiE_3Y2"}
	PhiE_3Y2 AT %Q* : UINT;
END_STRUCT
END_TYPE

// ---- DUTs/IO/PDOs/APS_Comm_Outputs_082002A4.TcDUT
{attribute 'GeneratedUsingTerminal: APS4322-7000-0017'}
{attribute addProperty BoxType "APS4322-7000-0017"}
{attribute addProperty Id "CommControlWordAT %Q*UINT2Data_1AT %Q*UINT2"}
{attribute addProperty CRC "136315556"}
{attribute addProperty Size "4"}
TYPE APS_Comm_Outputs_082002A4 EXTENDS OutputBase_10CEE7DE :
STRUCT
	{attribute addProperty Name "CommControlWord"}
	CommControlWord AT %Q* : UINT;
	{attribute addProperty Name "Data_1"}
	Data_1 AT %Q* : UINT;
END_STRUCT
END_TYPE

// ---- DUTs/IO/PDOs/InfoData_E68C61CD.TcDUT
{attribute 'GeneratedUsingTerminal: IODEVICETYPE_ETHERCATPROT'}
{attribute addProperty BoxType "IODEVICETYPE_ETHERCATPROT"}
{attribute addProperty Id "ChangeCountAT %I*UINT2DevIdAT %I*UINT2AmsNetIdAT %I*AMSNETID6CfgSlaveCountAT %I*UINT2DcToTcTimeOffsetAT %I*LINT8DcToExtTimeOffsetAT %I*LINT8"}
{attribute addProperty CRC "3867959757"}
{attribute addProperty Size "28"}
TYPE InfoData_E68C61CD EXTENDS InputBase_8311D824 :
STRUCT
	{attribute addProperty Name "ChangeCount"}
	ChangeCount AT %I* : UINT;
	{attribute addProperty Name "DevId"}
	DevId AT %I* : UINT;
	{attribute addProperty Name "AmsNetId"}
	AmsNetId AT %I* : AMSNETID;
	{attribute addProperty Name "CfgSlaveCount"}
	CfgSlaveCount AT %I* : UINT;
	{attribute addProperty Name "DcToTcTimeOffset"}
	DcToTcTimeOffset AT %I* : LINT;
	{attribute addProperty Name "DcToExtTimeOffset"}
	DcToExtTimeOffset AT %I* : LINT;
END_STRUCT
END_TYPE

// ---- DUTs/IO/PDOs/WcState_0B2B16F9.TcDUT
{attribute 'GeneratedUsingTerminal: IODEVICETYPE_ETHERCATPROT'}
{attribute addProperty BoxType "IODEVICETYPE_ETHERCATPROT"}
{attribute addProperty Id "WcStateAT %I*BOOL1"}
{attribute addProperty CRC "187373305"}
{attribute addProperty Size "1"}
TYPE WcState_0B2B16F9 :
STRUCT
	{attribute addProperty Name "WcState"}
	WcState AT %I* : BOOL;
END_STRUCT
END_TYPE

// ---- DUTs/IO/PDOs/InfoData_2A97D6CF.TcDUT
{attribute 'GeneratedUsingTerminal: IODEVICETYPE_ETHERCATPROT'}
{attribute addProperty BoxType "IODEVICETYPE_ETHERCATPROT"}
{attribute addProperty Id "ObjectIdAT %I*OTCID4StateAT %I*UINT2SlaveCountAT %I*UINT2"}
{attribute addProperty CRC "714593999"}
{attribute addProperty Size "8"}
TYPE InfoData_2A97D6CF EXTENDS InputBase_8311D824 :
STRUCT
	{attribute addProperty Name "ObjectId"}
	ObjectId AT %I* : OTCID;
	{attribute addProperty Name "State"}
	State AT %I* : UINT;
	{attribute addProperty Name "SlaveCount"}
	SlaveCount AT %I* : UINT;
END_STRUCT
END_TYPE

// ---- DUTs/IO/PDOs/Inputs_25A0042B.TcDUT
{attribute 'GeneratedUsingTerminal: IODEVICETYPE_ETHERCATPROT'}
{attribute addProperty BoxType "IODEVICETYPE_ETHERCATPROT"}
{attribute addProperty Id "SlaveCountAT %I*UINT2DevStateAT %I*UINT2Frm0StateAT %I*UINT2Frm0WcStateAT %I*UINT2Frm0InputToggleAT %I*UINT2Frm1StateAT %I*UINT2Frm1WcStateAT %I*UINT2Frm1InputToggleAT %I*UINT2Frm2StateAT %I*UINT2Frm2WcStateAT %I*UINT2Frm2InputToggleAT %I*UINT2Frm3StateAT %I*UINT2Frm3WcStateAT %I*UINT2Frm3InputToggleAT %I*UINT2Frm4StateAT %I*UINT2Frm4WcStateAT %I*UINT2Frm4InputToggleAT %I*UINT2Frm5StateAT %I*UINT2Frm5WcStateAT %I*UINT2Frm5InputToggleAT %I*UINT2Frm6StateAT %I*UINT2Frm6WcStateAT %I*UINT2Frm6InputToggleAT %I*UINT2Frm7StateAT %I*UINT2Frm7WcStateAT %I*UINT2Frm7InputToggleAT %I*UINT2Frm8StateAT %I*UINT2Frm8WcStateAT %I*UINT2Frm8InputToggleAT %I*UINT2Frm9StateAT %I*UINT2Frm9WcStateAT %I*UINT2Frm9InputToggleAT %I*UINT2Frm10StateAT %I*UINT2Frm10WcStateAT %I*UINT2Frm10InputToggleAT %I*UINT2Frm11StateAT %I*UINT2Frm11WcStateAT %I*UINT2Frm11InputToggleAT %I*UINT2Frm12StateAT %I*UINT2Frm12WcStateAT %I*UINT2Frm12InputToggleAT %I*UINT2Frm13StateAT %I*UINT2Frm13WcStateAT %I*UINT2Frm13InputToggleAT %I*UINT2Frm14StateAT %I*UINT2Frm14WcStateAT %I*UINT2Frm14InputToggleAT %I*UINT2Frm15StateAT %I*UINT2Frm15WcStateAT %I*UINT2Frm15InputToggleAT %I*UINT2Frm16StateAT %I*UINT2Frm16WcStateAT %I*UINT2Frm16InputToggleAT %I*UINT2Frm17StateAT %I*UINT2Frm17WcStateAT %I*UINT2Frm17InputToggleAT %I*UINT2Frm18StateAT %I*UINT2Frm18WcStateAT %I*UINT2Frm18InputToggleAT %I*UINT2Frm19StateAT %I*UINT2Frm19WcStateAT %I*UINT2Frm19InputToggleAT %I*UINT2Frm20StateAT %I*UINT2Frm20WcStateAT %I*UINT2Frm20InputToggleAT %I*UINT2Frm21StateAT %I*UINT2Frm21WcStateAT %I*UINT2Frm21InputToggleAT %I*UINT2Frm22StateAT %I*UINT2Frm22WcStateAT %I*UINT2Frm22InputToggleAT %I*UINT2Frm23StateAT %I*UINT2Frm23WcStateAT %I*UINT2Frm23InputToggleAT %I*UINT2Frm24StateAT %I*UINT2Frm24WcStateAT %I*UINT2Frm24InputToggleAT %I*UINT2Frm25StateAT %I*UINT2Frm25WcStateAT %I*UINT2Frm25InputToggleAT %I*UINT2"}
{attribute addProperty CRC "631243819"}
{attribute addProperty Size "160"}
TYPE Inputs_25A0042B EXTENDS InputBase_8311D824 :
STRUCT
	{attribute addProperty Name "SlaveCount"}
	SlaveCount AT %I* : UINT;
	{attribute addProperty Name "DevState"}
	DevState AT %I* : UINT;
	{attribute addProperty Name "Frm0State"}
	Frm0State AT %I* : UINT;
	{attribute addProperty Name "Frm0WcState"}
	Frm0WcState AT %I* : UINT;
	{attribute addProperty Name "Frm0InputToggle"}
	Frm0InputToggle AT %I* : UINT;
	{attribute addProperty Name "Frm1State"}
	Frm1State AT %I* : UINT;
	{attribute addProperty Name "Frm1WcState"}
	Frm1WcState AT %I* : UINT;
	{attribute addProperty Name "Frm1InputToggle"}
	Frm1InputToggle AT %I* : UINT;
	{attribute addProperty Name "Frm2State"}
	Frm2State AT %I* : UINT;
	{attribute addProperty Name "Frm2WcState"}
	Frm2WcState AT %I* : UINT;
	{attribute addProperty Name "Frm2InputToggle"}
	Frm2InputToggle AT %I* : UINT;
	{attribute addProperty Name "Frm3State"}
	Frm3State AT %I* : UINT;
	{attribute addProperty Name "Frm3WcState"}
	Frm3WcState AT %I* : UINT;
	{attribute addProperty Name "Frm3InputToggle"}
	Frm3InputToggle AT %I* : UINT;
	{attribute addProperty Name "Frm4State"}
	Frm4State AT %I* : UINT;
	{attribute addProperty Name "Frm4WcState"}
	Frm4WcState AT %I* : UINT;
	{attribute addProperty Name "Frm4InputToggle"}
	Frm4InputToggle AT %I* : UINT;
	{attribute addProperty Name "Frm5State"}
	Frm5State AT %I* : UINT;
	{attribute addProperty Name "Frm5WcState"}
	Frm5WcState AT %I* : UINT;
	{attribute addProperty Name "Frm5InputToggle"}
	Frm5InputToggle AT %I* : UINT;
	{attribute addProperty Name "Frm6State"}
	Frm6State AT %I* : UINT;
	{attribute addProperty Name "Frm6WcState"}
	Frm6WcState AT %I* : UINT;
	{attribute addProperty Name "Frm6InputToggle"}
	Frm6InputToggle AT %I* : UINT;
	{attribute addProperty Name "Frm7State"}
	Frm7State AT %I* : UINT;
	{attribute addProperty Name "Frm7WcState"}
	Frm7WcState AT %I* : UINT;
	{attribute addProperty Name "Frm7InputToggle"}
	Frm7InputToggle AT %I* : UINT;
	{attribute addProperty Name "Frm8State"}
	Frm8State AT %I* : UINT;
	{attribute addProperty Name "Frm8WcState"}
	Frm8WcState AT %I* : UINT;
	{attribute addProperty Name "Frm8InputToggle"}
	Frm8InputToggle AT %I* : UINT;
	{attribute addProperty Name "Frm9State"}
	Frm9State AT %I* : UINT;
	{attribute addProperty Name "Frm9WcState"}
	Frm9WcState AT %I* : UINT;
	{attribute addProperty Name "Frm9InputToggle"}
	Frm9InputToggle AT %I* : UINT;
	{attribute addProperty Name "Frm10State"}
	Frm10State AT %I* : UINT;
	{attribute addProperty Name "Frm10WcState"}
	Frm10WcState AT %I* : UINT;
	{attribute addProperty Name "Frm10InputToggle"}
	Frm10InputToggle AT %I* : UINT;
	{attribute addProperty Name "Frm11State"}
	Frm11State AT %I* : UINT;
	{attribute addProperty Name "Frm11WcState"}
	Frm11WcState AT %I* : UINT;
	{attribute addProperty Name "Frm11InputToggle"}
	Frm11InputToggle AT %I* : UINT;
	{attribute addProperty Name "Frm12State"}
	Frm12State AT %I* : UINT;
	{attribute addProperty Name "Frm12WcState"}
	Frm12WcState AT %I* : UINT;
	{attribute addProperty Name "Frm12InputToggle"}
	Frm12InputToggle AT %I* : UINT;
	{attribute addProperty Name "Frm13State"}
	Frm13State AT %I* : UINT;
	{attribute addProperty Name "Frm13WcState"}
	Frm13WcState AT %I* : UINT;
	{attribute addProperty Name "Frm13InputToggle"}
	Frm13InputToggle AT %I* : UINT;
	{attribute addProperty Name "Frm14State"}
	Frm14State AT %I* : UINT;
	{attribute addProperty Name "Frm14WcState"}
	Frm14WcState AT %I* : UINT;
	{attribute addProperty Name "Frm14InputToggle"}
	Frm14InputToggle AT %I* : UINT;
	{attribute addProperty Name "Frm15State"}
	Frm15State AT %I* : UINT;
	{attribute addProperty Name "Frm15WcState"}
	Frm15WcState AT %I* : UINT;
	{attribute addProperty Name "Frm15InputToggle"}
	Frm15InputToggle AT %I* : UINT;
	{attribute addProperty Name "Frm16State"}
	Frm16State AT %I* : UINT;
	{attribute addProperty Name "Frm16WcState"}
	Frm16WcState AT %I* : UINT;
	{attribute addProperty Name "Frm16InputToggle"}
	Frm16InputToggle AT %I* : UINT;
	{attribute addProperty Name "Frm17State"}
	Frm17State AT %I* : UINT;
	{attribute addProperty Name "Frm17WcState"}
	Frm17WcState AT %I* : UINT;
	{attribute addProperty Name "Frm17InputToggle"}
	Frm17InputToggle AT %I* : UINT;
	{attribute addProperty Name "Frm18State"}
	Frm18State AT %I* : UINT;
	{attribute addProperty Name "Frm18WcState"}
	Frm18WcState AT %I* : UINT;
	{attribute addProperty Name "Frm18InputToggle"}
	Frm18InputToggle AT %I* : UINT;
	{attribute addProperty Name "Frm19State"}
	Frm19State AT %I* : UINT;
	{attribute addProperty Name "Frm19WcState"}
	Frm19WcState AT %I* : UINT;
	{attribute addProperty Name "Frm19InputToggle"}
	Frm19InputToggle AT %I* : UINT;
	{attribute addProperty Name "Frm20State"}
	Frm20State AT %I* : UINT;
	{attribute addProperty Name "Frm20WcState"}
	Frm20WcState AT %I* : UINT;
	{attribute addProperty Name "Frm20InputToggle"}
	Frm20InputToggle AT %I* : UINT;
	{attribute addProperty Name "Frm21State"}
	Frm21State AT %I* : UINT;
	{attribute addProperty Name "Frm21WcState"}
	Frm21WcState AT %I* : UINT;
	{attribute addProperty Name "Frm21InputToggle"}
	Frm21InputToggle AT %I* : UINT;
	{attribute addProperty Name "Frm22State"}
	Frm22State AT %I* : UINT;
	{attribute addProperty Name "Frm22WcState"}
	Frm22WcState AT %I* : UINT;
	{attribute addProperty Name "Frm22InputToggle"}
	Frm22InputToggle AT %I* : UINT;
	{attribute addProperty Name "Frm23State"}
	Frm23State AT %I* : UINT;
	{attribute addProperty Name "Frm23WcState"}
	Frm23WcState AT %I* : UINT;
	{attribute addProperty Name "Frm23InputToggle"}
	Frm23InputToggle AT %I* : UINT;
	{attribute addProperty Name "Frm24State"}
	Frm24State AT %I* : UINT;
	{attribute addProperty Name "Frm24WcState"}
	Frm24WcState AT %I* : UINT;
	{attribute addProperty Name "Frm24InputToggle"}
	Frm24InputToggle AT %I* : UINT;
	{attribute addProperty Name "Frm25State"}
	Frm25State AT %I* : UINT;
	{attribute addProperty Name "Frm25WcState"}
	Frm25WcState AT %I* : UINT;
	{attribute addProperty Name "Frm25InputToggle"}
	Frm25InputToggle AT %I* : UINT;
END_STRUCT
END_TYPE

// ---- DUTs/IO/PDOs/Outputs_2397A10E.TcDUT
{attribute 'GeneratedUsingTerminal: IODEVICETYPE_ETHERCATPROT'}
{attribute addProperty BoxType "IODEVICETYPE_ETHERCATPROT"}
{attribute addProperty Id "DevCtrlAT %Q*UINT2Frm0CtrlAT %Q*UINT2Frm0WcCtrlAT %Q*UINT2Frm1CtrlAT %Q*UINT2Frm1WcCtrlAT %Q*UINT2Frm2CtrlAT %Q*UINT2Frm2WcCtrlAT %Q*UINT2Frm3CtrlAT %Q*UINT2Frm3WcCtrlAT %Q*UINT2Frm4CtrlAT %Q*UINT2Frm4WcCtrlAT %Q*UINT2Frm5CtrlAT %Q*UINT2Frm5WcCtrlAT %Q*UINT2Frm6CtrlAT %Q*UINT2Frm6WcCtrlAT %Q*UINT2Frm7CtrlAT %Q*UINT2Frm7WcCtrlAT %Q*UINT2Frm8CtrlAT %Q*UINT2Frm8WcCtrlAT %Q*UINT2Frm9CtrlAT %Q*UINT2Frm9WcCtrlAT %Q*UINT2Frm10CtrlAT %Q*UINT2Frm10WcCtrlAT %Q*UINT2Frm11CtrlAT %Q*UINT2Frm11WcCtrlAT %Q*UINT2Frm12CtrlAT %Q*UINT2Frm12WcCtrlAT %Q*UINT2Frm13CtrlAT %Q*UINT2Frm13WcCtrlAT %Q*UINT2Frm14CtrlAT %Q*UINT2Frm14WcCtrlAT %Q*UINT2Frm15CtrlAT %Q*UINT2Frm15WcCtrlAT %Q*UINT2Frm16CtrlAT %Q*UINT2Frm16WcCtrlAT %Q*UINT2Frm17CtrlAT %Q*UINT2Frm17WcCtrlAT %Q*UINT2Frm18CtrlAT %Q*UINT2Frm18WcCtrlAT %Q*UINT2Frm19CtrlAT %Q*UINT2Frm19WcCtrlAT %Q*UINT2Frm20CtrlAT %Q*UINT2Frm20WcCtrlAT %Q*UINT2Frm21CtrlAT %Q*UINT2Frm21WcCtrlAT %Q*UINT2Frm22CtrlAT %Q*UINT2Frm22WcCtrlAT %Q*UINT2Frm23CtrlAT %Q*UINT2Frm23WcCtrlAT %Q*UINT2Frm24CtrlAT %Q*UINT2Frm24WcCtrlAT %Q*UINT2Frm25CtrlAT %Q*UINT2Frm25WcCtrlAT %Q*UINT2"}
{attribute addProperty CRC "597139726"}
{attribute addProperty Size "106"}
TYPE Outputs_2397A10E EXTENDS OutputBase_10CEE7DE :
STRUCT
	{attribute addProperty Name "DevCtrl"}
	DevCtrl AT %Q* : UINT;
	{attribute addProperty Name "Frm0Ctrl"}
	Frm0Ctrl AT %Q* : UINT;
	{attribute addProperty Name "Frm0WcCtrl"}
	Frm0WcCtrl AT %Q* : UINT;
	{attribute addProperty Name "Frm1Ctrl"}
	Frm1Ctrl AT %Q* : UINT;
	{attribute addProperty Name "Frm1WcCtrl"}
	Frm1WcCtrl AT %Q* : UINT;
	{attribute addProperty Name "Frm2Ctrl"}
	Frm2Ctrl AT %Q* : UINT;
	{attribute addProperty Name "Frm2WcCtrl"}
	Frm2WcCtrl AT %Q* : UINT;
	{attribute addProperty Name "Frm3Ctrl"}
	Frm3Ctrl AT %Q* : UINT;
	{attribute addProperty Name "Frm3WcCtrl"}
	Frm3WcCtrl AT %Q* : UINT;
	{attribute addProperty Name "Frm4Ctrl"}
	Frm4Ctrl AT %Q* : UINT;
	{attribute addProperty Name "Frm4WcCtrl"}
	Frm4WcCtrl AT %Q* : UINT;
	{attribute addProperty Name "Frm5Ctrl"}
	Frm5Ctrl AT %Q* : UINT;
	{attribute addProperty Name "Frm5WcCtrl"}
	Frm5WcCtrl AT %Q* : UINT;
	{attribute addProperty Name "Frm6Ctrl"}
	Frm6Ctrl AT %Q* : UINT;
	{attribute addProperty Name "Frm6WcCtrl"}
	Frm6WcCtrl AT %Q* : UINT;
	{attribute addProperty Name "Frm7Ctrl"}
	Frm7Ctrl AT %Q* : UINT;
	{attribute addProperty Name "Frm7WcCtrl"}
	Frm7WcCtrl AT %Q* : UINT;
	{attribute addProperty Name "Frm8Ctrl"}
	Frm8Ctrl AT %Q* : UINT;
	{attribute addProperty Name "Frm8WcCtrl"}
	Frm8WcCtrl AT %Q* : UINT;
	{attribute addProperty Name "Frm9Ctrl"}
	Frm9Ctrl AT %Q* : UINT;
	{attribute addProperty Name "Frm9WcCtrl"}
	Frm9WcCtrl AT %Q* : UINT;
	{attribute addProperty Name "Frm10Ctrl"}
	Frm10Ctrl AT %Q* : UINT;
	{attribute addProperty Name "Frm10WcCtrl"}
	Frm10WcCtrl AT %Q* : UINT;
	{attribute addProperty Name "Frm11Ctrl"}
	Frm11Ctrl AT %Q* : UINT;
	{attribute addProperty Name "Frm11WcCtrl"}
	Frm11WcCtrl AT %Q* : UINT;
	{attribute addProperty Name "Frm12Ctrl"}
	Frm12Ctrl AT %Q* : UINT;
	{attribute addProperty Name "Frm12WcCtrl"}
	Frm12WcCtrl AT %Q* : UINT;
	{attribute addProperty Name "Frm13Ctrl"}
	Frm13Ctrl AT %Q* : UINT;
	{attribute addProperty Name "Frm13WcCtrl"}
	Frm13WcCtrl AT %Q* : UINT;
	{attribute addProperty Name "Frm14Ctrl"}
	Frm14Ctrl AT %Q* : UINT;
	{attribute addProperty Name "Frm14WcCtrl"}
	Frm14WcCtrl AT %Q* : UINT;
	{attribute addProperty Name "Frm15Ctrl"}
	Frm15Ctrl AT %Q* : UINT;
	{attribute addProperty Name "Frm15WcCtrl"}
	Frm15WcCtrl AT %Q* : UINT;
	{attribute addProperty Name "Frm16Ctrl"}
	Frm16Ctrl AT %Q* : UINT;
	{attribute addProperty Name "Frm16WcCtrl"}
	Frm16WcCtrl AT %Q* : UINT;
	{attribute addProperty Name "Frm17Ctrl"}
	Frm17Ctrl AT %Q* : UINT;
	{attribute addProperty Name "Frm17WcCtrl"}
	Frm17WcCtrl AT %Q* : UINT;
	{attribute addProperty Name "Frm18Ctrl"}
	Frm18Ctrl AT %Q* : UINT;
	{attribute addProperty Name "Frm18WcCtrl"}
	Frm18WcCtrl AT %Q* : UINT;
	{attribute addProperty Name "Frm19Ctrl"}
	Frm19Ctrl AT %Q* : UINT;
	{attribute addProperty Name "Frm19WcCtrl"}
	Frm19WcCtrl AT %Q* : UINT;
	{attribute addProperty Name "Frm20Ctrl"}
	Frm20Ctrl AT %Q* : UINT;
	{attribute addProperty Name "Frm20WcCtrl"}
	Frm20WcCtrl AT %Q* : UINT;
	{attribute addProperty Name "Frm21Ctrl"}
	Frm21Ctrl AT %Q* : UINT;
	{attribute addProperty Name "Frm21WcCtrl"}
	Frm21WcCtrl AT %Q* : UINT;
	{attribute addProperty Name "Frm22Ctrl"}
	Frm22Ctrl AT %Q* : UINT;
	{attribute addProperty Name "Frm22WcCtrl"}
	Frm22WcCtrl AT %Q* : UINT;
	{attribute addProperty Name "Frm23Ctrl"}
	Frm23Ctrl AT %Q* : UINT;
	{attribute addProperty Name "Frm23WcCtrl"}
	Frm23WcCtrl AT %Q* : UINT;
	{attribute addProperty Name "Frm24Ctrl"}
	Frm24Ctrl AT %Q* : UINT;
	{attribute addProperty Name "Frm24WcCtrl"}
	Frm24WcCtrl AT %Q* : UINT;
	{attribute addProperty Name "Frm25Ctrl"}
	Frm25Ctrl AT %Q* : UINT;
	{attribute addProperty Name "Frm25WcCtrl"}
	Frm25WcCtrl AT %Q* : UINT;
END_STRUCT
END_TYPE

// ---- DUTs/IO/Boxes/EK1100_1FC0878B.TcDUT
{attribute 'GeneratedUsingTerminal: EK1100-0000-0018'}
{attribute addProperty BoxType "EK1100-0000-0018"}
{attribute addProperty Description "EK1100 EtherCAT Coupler (2A E-Bus)"}
{attribute addProperty Physics "YKY"}
{attribute addProperty Id "InfoDataAT %I*InfoData_6F19DB2B2"}
{attribute addProperty CRC "532711307"}
{attribute addProperty Size "2"}
TYPE EK1100_1FC0878B EXTENDS EtcSlaveBoxBase_77A0E4A7 :
STRUCT
	{attribute addProperty Name "InfoData"}
	InfoData : InfoData_6F19DB2B;
END_STRUCT
END_TYPE

// ---- DUTs/IO/Boxes/EK1122_1FC0878B.TcDUT
{attribute 'GeneratedUsingTerminal: EK1122-0000-0018'}
{attribute addProperty BoxType "EK1122-0000-0018"}
{attribute addProperty Description "EK1122 2 port EtherCAT junction"}
{attribute addProperty Physics "KYKY"}
{attribute addProperty Id "InfoDataAT %I*InfoData_6F19DB2B2"}
{attribute addProperty CRC "532711307"}
{attribute addProperty Size "2"}
TYPE EK1122_1FC0878B EXTENDS EtcSlaveTerminalBase_947E5A46 :
STRUCT
	{attribute addProperty Name "InfoData"}
	InfoData : InfoData_6F19DB2B;
END_STRUCT
END_TYPE

// ---- DUTs/IO/Boxes/APS1003_C6D7567B.TcDUT
{attribute 'GeneratedUsingTerminal: APS1003-7000-0016'}
{attribute addProperty BoxType "APS1003-7000-0016"}
{attribute addProperty Description "APS1003-7000 Drive"}
{attribute addProperty Physics "YKY"}
{attribute addProperty Id "YVR_InputsAT %I*YVR_Inputs_4719D0DB98YVR_OutputsAT %Q*YVR_Outputs_31F2CBB3146WcStateAT %I*WcState_9091E0EB2InfoDataAT %I*InfoData_BEF6B88E18"}
{attribute addProperty CRC "3336001147"}
{attribute addProperty Size "264"}
TYPE APS1003_C6D7567B EXTENDS EtcSlaveBoxBase_77A0E4A7 :
STRUCT
	{attribute addProperty Name "YVR_Inputs"}
	YVR_Inputs : YVR_Inputs_4719D0DB;
	{attribute addProperty Name "YVR_Outputs"}
	YVR_Outputs : YVR_Outputs_31F2CBB3;
	{attribute addProperty Name "WcState"}
	WcState : WcState_9091E0EB;
	{attribute addProperty Name "InfoData"}
	InfoData : InfoData_BEF6B88E;
END_STRUCT
END_TYPE

// ---- DUTs/IO/Boxes/APS1003_A49C5437.TcDUT
{attribute 'GeneratedUsingTerminal: APS1003-5000-0016'}
{attribute addProperty BoxType "APS1003-5000-0016"}
{attribute addProperty Description "APS1003-5000 Feedback"}
{attribute addProperty Physics "K"}
{attribute addProperty Id "FB_InputsAT %I*FB_Inputs_F0F03BDD308WcStateAT %I*WcState_9091E0EB2InfoDataAT %I*InfoData_A7436BC610"}
{attribute addProperty CRC "2761708599"}
{attribute addProperty Size "320"}
TYPE APS1003_A49C5437 EXTENDS EtcSlaveTerminalBase_947E5A46 :
STRUCT
	{attribute addProperty Name "FB_Inputs"}
	FB_Inputs : FB_Inputs_F0F03BDD;
	{attribute addProperty Name "WcState"}
	WcState : WcState_9091E0EB;
	{attribute addProperty Name "InfoData"}
	InfoData : InfoData_A7436BC6;
END_STRUCT
END_TYPE

// ---- DUTs/IO/Boxes/APS4322_7CC84994.TcDUT
{attribute 'GeneratedUsingTerminal: APS4322-7000-0017'}
{attribute addProperty BoxType "APS4322-7000-0017"}
{attribute addProperty Description "APS4322-7000 Drive"}
{attribute addProperty Physics "YKY"}
{attribute addProperty Id "APS_InputsAT %I*APS_Inputs_4719D0DB98APS_DiagdataAT %I*APS_Diagdata_CE5B986F4APS_Comm_InputsAT %I*APS_Comm_Inputs_388FE28E10APS_OutputsAT %Q*APS_Outputs_31F2CBB3146APS_Comm_OutputsAT %Q*APS_Comm_Outputs_082002A44WcStateAT %I*WcState_9091E0EB2InfoDataAT %I*InfoData_BEF6B88E18"}
{attribute addProperty CRC "2093500820"}
{attribute addProperty Size "282"}
TYPE APS4322_7CC84994 EXTENDS EtcSlaveBoxBase_77A0E4A7 :
STRUCT
	{attribute addProperty Name "APS_Inputs"}
	APS_Inputs : APS_Inputs_4719D0DB;
	{attribute addProperty Name "APS_Diagdata"}
	APS_Diagdata : APS_Diagdata_CE5B986F;
	{attribute addProperty Name "APS_Comm_Inputs"}
	APS_Comm_Inputs : APS_Comm_Inputs_388FE28E;
	{attribute addProperty Name "APS_Outputs"}
	APS_Outputs : APS_Outputs_31F2CBB3;
	{attribute addProperty Name "APS_Comm_Outputs"}
	APS_Comm_Outputs : APS_Comm_Outputs_082002A4;
	{attribute addProperty Name "WcState"}
	WcState : WcState_9091E0EB;
	{attribute addProperty Name "InfoData"}
	InfoData : InfoData_BEF6B88E;
END_STRUCT
END_TYPE

// ---- DUTs/IO/Boxes/APS4322_A49C5437.TcDUT
{attribute 'GeneratedUsingTerminal: APS4322-5000-0017'}
{attribute addProperty BoxType "APS4322-5000-0017"}
{attribute addProperty Description "APS4322-5000 Feedback"}
{attribute addProperty Physics "K"}
{attribute addProperty Id "FB_InputsAT %I*FB_Inputs_F0F03BDD308WcStateAT %I*WcState_9091E0EB2InfoDataAT %I*InfoData_A7436BC610"}
{attribute addProperty CRC "2761708599"}
{attribute addProperty Size "320"}
TYPE APS4322_A49C5437 EXTENDS EtcSlaveTerminalBase_947E5A46 :
STRUCT
	{attribute addProperty Name "FB_Inputs"}
	FB_Inputs : FB_Inputs_F0F03BDD;
	{attribute addProperty Name "WcState"}
	WcState : WcState_9091E0EB;
	{attribute addProperty Name "InfoData"}
	InfoData : InfoData_A7436BC6;
END_STRUCT
END_TYPE

// ---- DUTs/IO/Devices/SyncUnitTask_2D604ED5.TcDUT
{attribute 'GeneratedUsingTerminal: IODEVICETYPE_ETHERCATPROT'}
{attribute addProperty BoxType "IODEVICETYPE_ETHERCATPROT"}
{attribute addProperty Id "WcStateAT %I*WcState_0B2B16F91InfoDataAT %I*InfoData_2A97D6CF8"}
{attribute addProperty CRC "761286357"}
{attribute addProperty Size "9"}
TYPE SyncUnitTask_2D604ED5 :
STRUCT
	{attribute addProperty Name "WcState"}
	WcState : WcState_0B2B16F9;
	{attribute addProperty Name "InfoData"}
	InfoData : InfoData_2A97D6CF;
END_STRUCT
END_TYPE

// ---- DUTs/IO/Devices/SyncUnitTasks_6FEB8257.TcDUT
{attribute 'GeneratedUsingTerminal: '}
{attribute addProperty BoxType ""}
{attribute addProperty Id "unreferencedAT %I*SyncUnitTask_2D604ED59PlcTaskAT %I*SyncUnitTask_2D604ED59"}
{attribute addProperty CRC "1877705303"}
{attribute addProperty Size "18"}
TYPE SyncUnitTasks_6FEB8257 :
STRUCT
	{attribute addProperty Name "unreferenced"}
	unreferenced : SyncUnitTask_2D604ED5;
	{attribute addProperty Name "PlcTask"}
	PlcTask : SyncUnitTask_2D604ED5;
END_STRUCT
END_TYPE

// ---- DUTs/IO/Devices/SyncUnits_99E584AF.TcDUT
{attribute 'GeneratedUsingTerminal: '}
{attribute addProperty BoxType ""}
{attribute addProperty Id "_defaultAT %I*SyncUnitTasks_6FEB825718"}
{attribute addProperty CRC "2581955759"}
{attribute addProperty Size "18"}
TYPE SyncUnits_99E584AF :
STRUCT
	{attribute addProperty Name "_default"}
	_default : SyncUnitTasks_6FEB8257;
END_STRUCT
END_TYPE

// ---- DUTs/IO/Topology/Beckhoff_APS1xxxEK1122_94631AF6.TcDUT
{attribute 'GeneratedUsingTerminal: EK1122-0000-0018'}
{attribute addProperty BoxType "EK1122-0000-0018"}
{attribute addProperty Id "Beckhoff_APS1xxxsub_EK1100EK1100_1FC0878B2A_0001_APS1003_7000_0016APS1003_C6D7567B264"}
{attribute addProperty CRC "2489522934"}
{attribute addProperty Size "266"}
{attribute addProperty Name "Beckhoff APS1xxxEK1122"}
TYPE Beckhoff_APS1xxxEK1122_94631AF6 EXTENDS EK1122_1FC0878B :
STRUCT
	{attribute addProperty Name "Beckhoff APS1xxxsub EK1100"}
	{attribute addProperty PreviousPort "Beckhoff APS1xxxEK1122 : D"}
	Beckhoff_APS1xxxsub_EK1100 : EK1100_1FC0878B;
	{attribute addProperty Name "A_0001(APS1003-7000-0016)"}
	{attribute addProperty PreviousPort "Beckhoff APS1xxxsub EK1100 : C"}
	A_0001_APS1003_7000_0016 : APS1003_C6D7567B;
END_STRUCT
END_TYPE

// ---- DUTs/IO/Topology/Beckhoff_APS1xxx_5C0D85AF.TcDUT
{attribute 'GeneratedUsingTerminal: EK1100-0000-0018'}
{attribute addProperty BoxType "EK1100-0000-0018"}
{attribute addProperty Id "Beckhoff_APS1xxxEK1122Beckhoff_APS1xxxEK1122_94631AF6266A_0002_APS1003_5000_0016APS1003_A49C5437320"}
{attribute addProperty CRC "1544390063"}
{attribute addProperty Size "586"}
{attribute addProperty Name "Beckhoff APS1xxx"}
TYPE Beckhoff_APS1xxx_5C0D85AF EXTENDS EK1100_1FC0878B :
STRUCT
	{attribute addProperty Name "Beckhoff APS1xxxEK1122"}
	{attribute addProperty PreviousPort "Beckhoff APS1xxx : B"}
	Beckhoff_APS1xxxEK1122 : Beckhoff_APS1xxxEK1122_94631AF6;
	{attribute addProperty Name "A_0002(APS1003-5000-0016)"}
	{attribute addProperty PreviousPort "Beckhoff APS1xxxEK1122 : C"}
	A_0002_APS1003_5000_0016 : APS1003_A49C5437;
END_STRUCT
END_TYPE

// ---- DUTs/IO/Topology/Beckhoff_APS4xxxEK1122_0B49C1F2.TcDUT
{attribute 'GeneratedUsingTerminal: EK1122-0000-0018'}
{attribute addProperty BoxType "EK1122-0000-0018"}
{attribute addProperty Id "Beckhoff_APS4xxxsub_EK1100EK1100_1FC0878B2A_0001_APS4322_7000_0017APS4322_7CC84994282"}
{attribute addProperty CRC "189383154"}
{attribute addProperty Size "284"}
{attribute addProperty Name "Beckhoff APS4xxxEK1122"}
TYPE Beckhoff_APS4xxxEK1122_0B49C1F2 EXTENDS EK1122_1FC0878B :
STRUCT
	{attribute addProperty Name "Beckhoff APS4xxxsub EK1100"}
	{attribute addProperty PreviousPort "Beckhoff APS4xxxEK1122 : D"}
	Beckhoff_APS4xxxsub_EK1100 : EK1100_1FC0878B;
	{attribute addProperty Name "A_0001(APS4322-7000-0017)"}
	{attribute addProperty PreviousPort "Beckhoff APS4xxxsub EK1100 : C"}
	A_0001_APS4322_7000_0017 : APS4322_7CC84994;
END_STRUCT
END_TYPE

// ---- DUTs/IO/Topology/Beckhoff_APS4xxx_9BEEA20F.TcDUT
{attribute 'GeneratedUsingTerminal: EK1100-0000-0018'}
{attribute addProperty BoxType "EK1100-0000-0018"}
{attribute addProperty Id "Beckhoff_APS4xxxEK1122Beckhoff_APS4xxxEK1122_0B49C1F2284A_0002_APS4322_5000_0017APS4322_A49C5437320"}
{attribute addProperty CRC "2616107535"}
{attribute addProperty Size "604"}
{attribute addProperty Name "Beckhoff APS4xxx"}
TYPE Beckhoff_APS4xxx_9BEEA20F EXTENDS EK1100_1FC0878B :
STRUCT
	{attribute addProperty Name "Beckhoff APS4xxxEK1122"}
	{attribute addProperty PreviousPort "Beckhoff APS4xxx : B"}
	Beckhoff_APS4xxxEK1122 : Beckhoff_APS4xxxEK1122_0B49C1F2;
	{attribute addProperty Name "A_0002(APS4322-5000-0017)"}
	{attribute addProperty PreviousPort "Beckhoff APS4xxxEK1122 : C"}
	A_0002_APS4322_5000_0017 : APS4322_A49C5437;
END_STRUCT
END_TYPE

// ---- DUTs/IO/Topology/EtherCAT_Master_APSxxxx_214E63DA.TcDUT
{attribute 'GeneratedUsingTerminal: IODEVICETYPE_ETHERCATPROT'}
{attribute addProperty BoxType "IODEVICETYPE_ETHERCATPROT"}
{attribute addProperty Id "Beckhoff_APS1xxxBeckhoff_APS1xxx_5C0D85AF586Beckhoff_APS4xxxBeckhoff_APS4xxx_9BEEA20F604SyncUnitsSyncUnits_99E584AF18InputsInputs_25A0042B160OutputsOutputs_2397A10E106InfoDataInfoData_E68C61CD28"}
{attribute addProperty CRC "558785498"}
{attribute addProperty Size "1502"}
{attribute addProperty Name "EtherCAT Master APSxxxx"}
TYPE EtherCAT_Master_APSxxxx_214E63DA EXTENDS EtcMasterBase_62654B43 :
STRUCT
	{attribute addProperty Name "Beckhoff APS1xxx"}
	{attribute addProperty PreviousPort "EtherCAT Master APSxxxx : Master"}
	Beckhoff_APS1xxx : Beckhoff_APS1xxx_5C0D85AF;
	{attribute addProperty Name "Beckhoff APS4xxx"}
	{attribute addProperty PreviousPort "Beckhoff APS1xxx : C"}
	Beckhoff_APS4xxx : Beckhoff_APS4xxx_9BEEA20F;
	{attribute addProperty Name "SyncUnits"}
	SyncUnits : SyncUnits_99E584AF;
	{attribute addProperty Name "Inputs"}
	Inputs : Inputs_25A0042B;
	{attribute addProperty Name "Outputs"}
	Outputs : Outputs_2397A10E;
	{attribute addProperty Name "InfoData"}
	InfoData : InfoData_E68C61CD;
END_STRUCT
END_TYPE

// ---- DUTs/IO/Base/EtcSlaveBase_82538BE2.TcDUT

TYPE EtcSlaveBase_82538BE2 :
STRUCT
END_STRUCT
END_TYPE

// ---- DUTs/IO/Base/EtcSlaveBase_82538BE2.TcDUT

TYPE EtcSlaveBase_82538BE2 :
STRUCT
END_STRUCT
END_TYPE

// ---- DUTs/IO/Base/EtcSlaveBase_82538BE2.TcDUT

TYPE EtcSlaveBase_82538BE2 :
STRUCT
END_STRUCT
END_TYPE

// ---- DUTs/IO/Base/EtcSlaveTerminalBase_947E5A46.TcDUT

{attribute clr[Container(Layout.Stack)]}
{attribute clr[Group(Layout.GroupBox)]}
{attribute addProperty PreviousPort "Unknown"}
TYPE EtcSlaveTerminalBase_947E5A46 EXTENDS EtcSlaveBase_82538BE2 :
STRUCT
END_STRUCT
END_TYPE

// ---- DUTs/IO/Base/EtcSlaveBoxBase_77A0E4A7.TcDUT

{attribute clr[Container(Layout.Stack)]}
{attribute clr[Group(Layout.GroupBox)]}
{attribute addProperty PreviousPort "Unknown"}
TYPE EtcSlaveBoxBase_77A0E4A7 EXTENDS EtcSlaveBase_82538BE2 :
STRUCT
END_STRUCT
END_TYPE

// ---- DUTs/IO/Base/EtcSlaveEndTerminalBase_866C7F0C.TcDUT

{attribute clr[Container(Layout.Stack)]}
{attribute clr[Group(Layout.GroupBox)]}
{attribute addProperty PreviousPort "Unknown"}
TYPE EtcSlaveEndTerminalBase_866C7F0C EXTENDS EtcSlaveBase_82538BE2 :
STRUCT
END_STRUCT
END_TYPE

// ---- DUTs/IO/Base/InputBase_8311D824.TcDUT

TYPE InputBase_8311D824 :
STRUCT
END_STRUCT
END_TYPE

// ---- DUTs/IO/Base/OutputBase_10CEE7DE.TcDUT

TYPE OutputBase_10CEE7DE :
STRUCT
END_STRUCT
END_TYPE

// ---- DUTs/IO/Base/EtcMasterBase_62654B43.TcDUT

TYPE EtcMasterBase_62654B43 :
STRUCT
END_STRUCT
END_TYPE

// ---- GVLs/GVL_iXlinker.TcGVL
{attribute 'qualified_only'}
VAR_GLOBAL
		EtherCAT_Master_APSxxxx : EtherCAT_Master_APSxxxx_214E63DA;
END_VAR

// ---- POUs/MAIN.TcPOU
PROGRAM MAIN
VAR
END_VAR

END_PROGRAM
